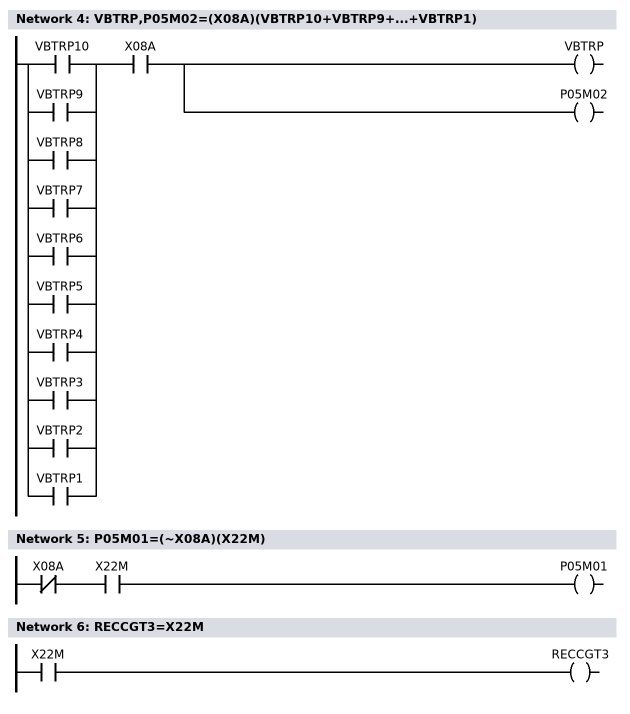
NETWORK
TITLE = VBTRP,P05M02=(X08A)(VBTRP10+VBTRP9+...+VBTRP1)
      A(;
      O     "VBTRP10";
      O     "VBTRP9";
      O     "VBTRP8";
      O     "VBTRP7";
      O     "VBTRP6";
      O     "VBTRP5";
      O     "VBTRP4";
      O     "VBTRP3";
      O     "VBTRP2";
      O     "VBTRP1";
      );
      A     "X08A";
      =     "VBTRP";
      =     "P05M02";
NETWORK
TITLE = P05M01=(~X08A)(X22M)
      AN    "X08A";
      A     "X22M";
      =     "P05M01";
NETWORK
TITLE = RECCGT3=X22M
      A     "X22M";
      =     "RECCGT3";
END_FUNCTION

FUNCTION "Sheet 22 (ATC)" : VOID	// FC 101
TITLE = Sheet 22 (ATC)
//LADDERS 32, 33, 41. VIBRATION RUNUP / RUNDOWN LOGIC (Digital)
AUTHOR : RJ
FAMILY : ATC
VERSION : 0.1
BEGIN
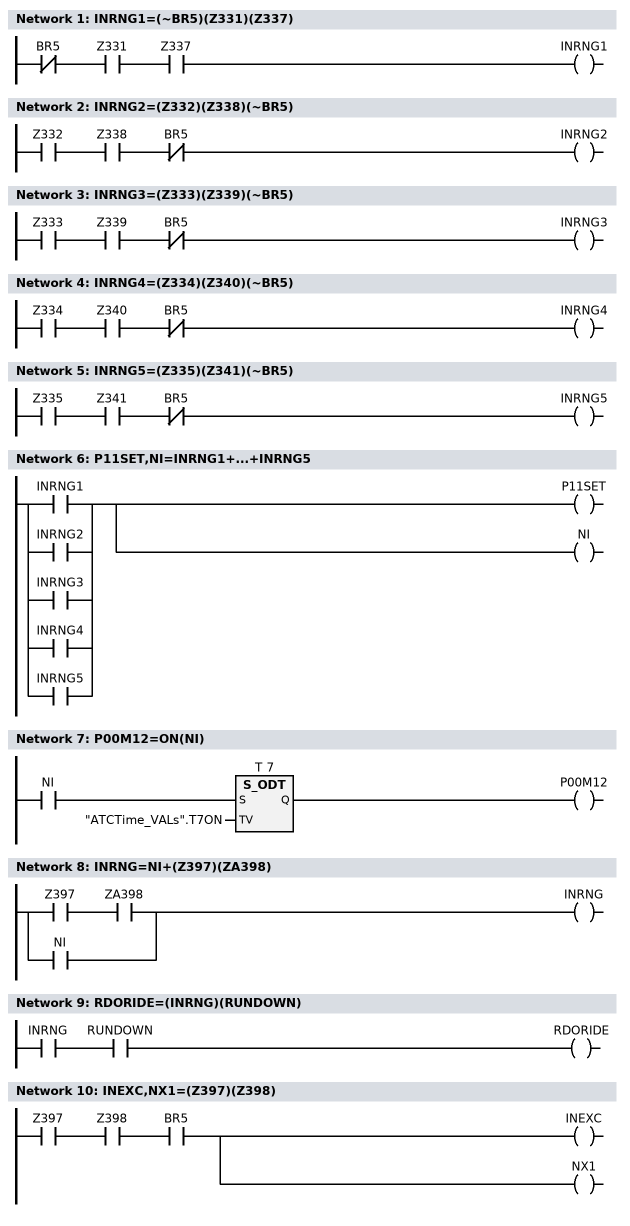
NETWORK
TITLE = INRNG1=(~BR5)(Z331)(Z337)
      AN    "BR5";
      A     "Z331";
      A     "Z337";
      =     "INRNG1";
NETWORK
TITLE = INRNG2=(Z332)(Z338)(~BR5)
      A     "Z332";
      A     "Z338";
      AN    "BR5";
      =     "INRNG2";
NETWORK
TITLE = INRNG3=(Z333)(Z339)(~BR5)
      A     "Z333";
      A     "Z339";
      AN    "BR5";
      =     "INRNG3";
NETWORK
TITLE = INRNG4=(Z334)(Z340)(~BR5)
      A     "Z334";
      A     "Z340";
      AN    "BR5";
      =     "INRNG4";
NETWORK
TITLE = INRNG5=(Z335)(Z341)(~BR5)
      A     "Z335";
      A     "Z341";
      AN    "BR5";
      =     "INRNG5";
NETWORK
TITLE = P11SET,NI=INRNG1+...+INRNG5
      O     "INRNG1";
      O     "INRNG2";
      O     "INRNG3";
      O     "INRNG4";
      O     "INRNG5";
      =     "P11SET";
      =     "NI";
NETWORK
TITLE = P00M12=ON(NI)
      A     "NI";
      L     "ATCTime_VALs".T7ON;
      SD    T 7;
      NOP   0;
      NOP   0;
      NOP   0;
      A     T 7;
      =     "P00M12";
NETWORK
TITLE = INRNG=NI+(Z397)(ZA398)
      A     "Z397";
      A     "ZA398";
      O     "NI";
      =     "INRNG";
NETWORK
TITLE = RDORIDE=(INRNG)(RUNDOWN)
      A     "INRNG";
      A     "RUNDOWN";
      =     "RDORIDE";
NETWORK
TITLE = INEXC,NX1=(Z397)(Z398)
      A     "Z397";
      A     "Z398";
      A     "BR5";
      =     "INEXC";
      =     "NX1";
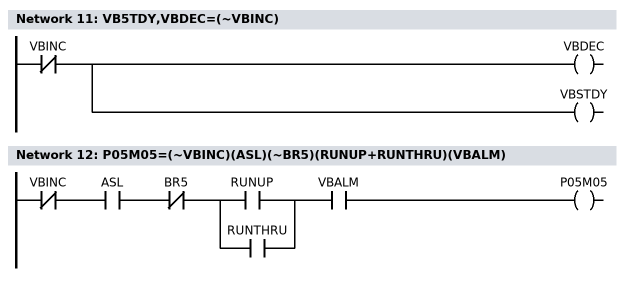
NETWORK
TITLE = VB5TDY,VBDEC=(~VBINC)
      AN    "VBINC";
      =     "VBDEC";
      =     "VBSTDY";
NETWORK
TITLE = P05M05=(~VBINC)(ASL)(~BR5)(RUNUP+RUNTHRU)(VBALM)
      AN    "VBINC";
      A     "ASL";
      AN    "BR5";
      A(;
      O     "RUNUP";
      O     "RUNTHRU";
      );
      A     "VBALM";
      =     "P05M05";
NETWORK
TITLE = HOLDSPD, HSOTIME
//HOLDSPD=FF[{(HSOTIME)(~INRNG)},{(~VBALM)+RUNUP+RUNTHRU+RUNDOWN+RUNBACK+VRSCNP}
//HSOTIME=FF{HOLSPD,(~VBALM)}
      A(;
      A     "HOLDSPD";
      S     "HSOTIME";
      AN    "VBALM";
      R     "HSOTIME";
      A     "HSOTIME";
      );
      AN    "INRNG";
      S     "HOLDSPD";
      A(;
      ON    "VBALM";
      O     "RUNUP";
      O     "RUNTHRU";
      O     "RUNDOWN";
      O     "RUNBACK";
      O     "VRSCNP";
      );
      R     "HOLDSPD";
      A     "HOLDSPD";
      =     "HOLDSPD";
END_FUNCTION

FUNCTION "Sheet 23 (ATC)" : VOID	// FC 102
TITLE = Sheet 23 (ATC)
//LADDER 39. VIBRATION RUNDOWN / RUNBACK LOGIC (Digital)
AUTHOR : RJ
FAMILY : ATC
VERSION : 0.1
BEGIN
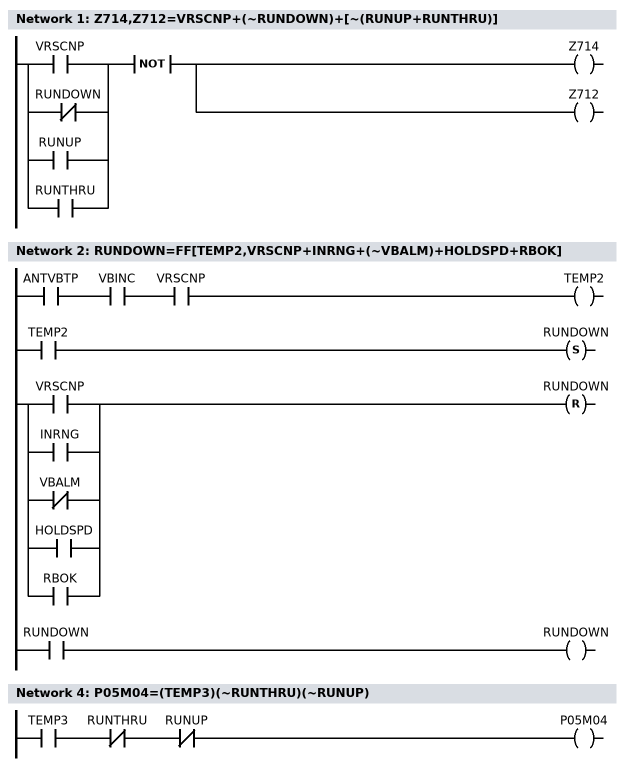
NETWORK
TITLE = Z714,Z712=VRSCNP+(~RUNDOWN)+[~(RUNUP+RUNTHRU)]
      O     "VRSCNP";
      ON    "RUNDOWN";
      O;
      A(;
      O     "RUNUP";
      O     "RUNTHRU";
      );
      NOT;
      =     "Z714";
      =     "Z712";
NETWORK
TITLE = RUNDOWN=FF[TEMP2,VRSCNP+INRNG+(~VBALM)+HOLDSPD+RBOK]
//TEMP2=(ANTVBTP)(VBINC)(VRSCNP)
      A     "ANTVBTP";
      A     "VBINC";
      A     "VRSCNP";
      =     "TEMP2";
      A     "TEMP2";
      S     "RUNDOWN";
      A(;
      O     "VRSCNP";
      O     "INRNG";
      ON    "VBALM";
      O     "HOLDSPD";
      O     "RBOK";
      );
      R     "RUNDOWN";
      A     "RUNDOWN";
      =     "RUNDOWN";
NETWORK
TITLE = RUNBACK, TEMP3
//RUNBACK=[(TEMP2)(~HOLDSPD)(RBOK)(~INRNG)(VBALM)]+FF[TEMP3,VRSCNP+RUNDOWN
//+RUNTHRU+RUNUP+(~RDEQASR)]
//TEMP3=RDORIDE+(HLDWS+VBALM+REQTRIP)(INEXC+INRNG)
      A     "TEMP2";
      AN    "HOLDSPD";
      A     "RBOK";
      AN    "INRNG";
      A     "VBALM";
      O(;
      A(;
      O     "RDORIDE";
      O;
      A(;
      O     "HLDWS";
      O     "VBALM";
      O     "REQTRIP";
      );
      A(;
      O     "INEXC";
      O     "INRNG";
      );
      );
      =     "TEMP3";
      A     "TEMP3";
      S     "TEMP4";
      A(;
      O     "VRSCNP";
      O     "RUNDOWN";
      O     "RUNTHRU";
      O     "RUNUP";
      ON    "RDEQASR";
      );
      R     "TEMP4";
      A     "TEMP4";
      );
      =     "RUNBACK";
NETWORK
TITLE = P05M04=(TEMP3)(~RUNTHRU)(~RUNUP)
      A     "TEMP3";
      AN    "RUNTHRU";
      AN    "RUNUP";
      =     "P05M04";
END_FUNCTION

FUNCTION "3xHISIGMTV, 1xLOSIGMTV" : VOID	// FC 103
TITLE = 3xHISIGMTV, 1xLOSIGMTV
AUTHOR : RJ
VERSION : 0.1
VAR_INPUT
  IN_HI1 : REAL ;
  IN_HI2 : REAL ;
  IN_HI3 : REAL ;
  IN_LO : REAL ;
  STPT : REAL ;
  Param_HI1 : UDT 8;
  Param_HI2 : UDT 8;
  Param_HI3 : UDT 8;
  Param_LO : UDT 9;
END_VAR
VAR_OUTPUT
  OUT_HI1 : BOOL ;
  OUT_HI2 : BOOL ;
  OUT_HI3 : BOOL ;
  OUT_LO : BOOL ;
END_VAR
VAR_TEMP
  TEMP_HI1 : UDT 8;
  TEMP_HI2 : UDT 8;
  TEMP_HI3 : UDT 8;
  TEMP_LO : UDT 9;
END_VAR
BEGIN
NETWORK
TITLE =
      BLD   5;
      T     LD 18;
      TAK;
      T     LD 22;
      L     P##Param_HI1;
      LAR1;
      L     W [AR1,P#0.0];
      T     LW 16;
      OPN   DB [LW 16];
      L     D [AR1,P#2.0];
      LAR1;
      L     LD 22;
      L     LD 18;
      L     D [AR1,P#0.0];
      T     #TEMP_HI1;
      NOP   0;
NETWORK
TITLE =
      BLD   5;
      T     LD 18;
      TAK;
      T     LD 22;
      L     P##Param_HI2;
      LAR1;
      L     W [AR1,P#0.0];
      T     LW 16;
      OPN   DB [LW 16];
      L     D [AR1,P#2.0];
      LAR1;
      L     LD 22;
      L     LD 18;
      L     D [AR1,P#0.0];
      T     #TEMP_HI2;
      NOP   0;
NETWORK
TITLE =
      BLD   5;
      T     LD 18;
      TAK;
      T     LD 22;
      L     P##Param_HI3;
      LAR1;
      L     W [AR1,P#0.0];
      T     LW 16;
      OPN   DB [LW 16];
      L     D [AR1,P#2.0];
      LAR1;
      L     LD 22;
      L     LD 18;
      L     D [AR1,P#0.0];
      T     #TEMP_HI3;
      NOP   0;
NETWORK
TITLE =
      BLD   5;
      T     LD 18;
      TAK;
      T     LD 22;
      L     P##Param_LO;
      LAR1;
      L     W [AR1,P#0.0];
      T     LW 16;
      OPN   DB [LW 16];
      L     D [AR1,P#2.0];
      LAR1;
      L     LD 22;
      L     LD 18;
      L     D [AR1,P#0.0];
      T     #TEMP_LO;
      NOP   0;
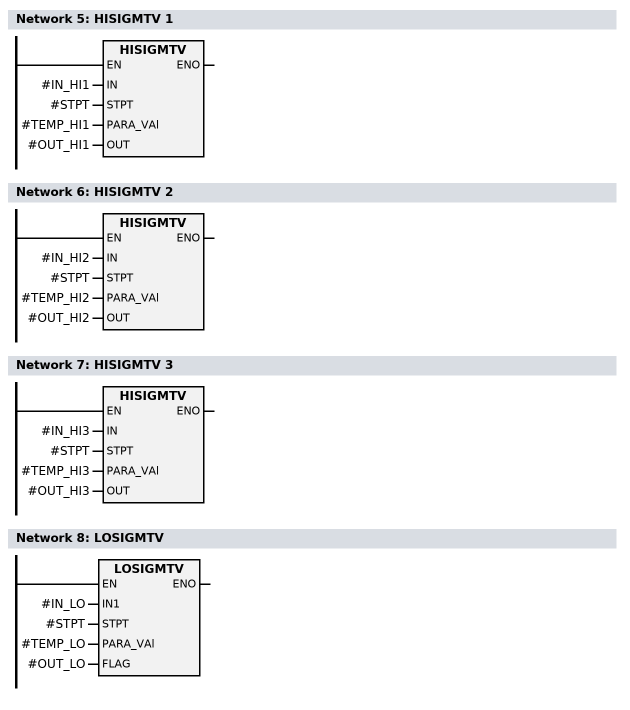
NETWORK
TITLE = HISIGMTV 1
      CALL  "HISIGMTV" (
           IN                       := #IN_HI1,
           STPT                     := #STPT,
           PARA_VAl                 := #TEMP_HI1,
           OUT                      := #OUT_HI1);
      NOP   0;
NETWORK
TITLE = HISIGMTV 2
      CALL  "HISIGMTV" (
           IN                       := #IN_HI2,
           STPT                     := #STPT,
           PARA_VAl                 := #TEMP_HI2,
           OUT                      := #OUT_HI2);
      NOP   0;
NETWORK
TITLE = HISIGMTV 3
      CALL  "HISIGMTV" (
           IN                       := #IN_HI3,
           STPT                     := #STPT,
           PARA_VAl                 := #TEMP_HI3,
           OUT                      := #OUT_HI3);
      NOP   0;
NETWORK
TITLE = LOSIGMTV
      CALL  "LOSIGMTV" (
           IN1                      := #IN_LO,
           STPT                     := #STPT,
           PARA_VAl                 := #TEMP_LO,
           FLAG                     := #OUT_LO);
      NOP   0;
END_FUNCTION

FUNCTION "3xLOSIGMTV, 1xHISIGMTV" : VOID	// FC 104
TITLE = 3xLOSIGMTV, 1xHISIGMTV
AUTHOR : RJ
VERSION : 0.1
VAR_INPUT
  IN_LO1 : REAL ;
  IN_LO2 : REAL ;
  IN_LO3 : REAL ;
  IN_HI : REAL ;
  STPT : REAL ;
  Param_LO1 : UDT 9;
  Param_LO2 : UDT 9;
  Param_LO3 : UDT 9;
  Param_HI : UDT 8;
END_VAR
VAR_OUTPUT
  OUT_LO1 : BOOL ;
  OUT_LO2 : BOOL ;
  OUT_LO3 : BOOL ;
  OUT_HI : BOOL ;
END_VAR
VAR_TEMP
  TEMP_LO1 : UDT 9;
  TEMP_LO2 : UDT 9;
  TEMP_LO3 : UDT 9;
  TEMP_HI : UDT 8;
END_VAR
BEGIN
NETWORK
TITLE =
      BLD   5;
      T     LD 18;
      TAK;
      T     LD 22;
      L     P##Param_LO1;
      LAR1;
      L     W [AR1,P#0.0];
      T     LW 16;
      OPN   DB [LW 16];
      L     D [AR1,P#2.0];
      LAR1;
      L     LD 22;
      L     LD 18;
      L     D [AR1,P#0.0];
      T     #TEMP_LO1;
      NOP   0;
NETWORK
TITLE =
      BLD   5;
      T     LD 18;
      TAK;
      T     LD 22;
      L     P##Param_LO2;
      LAR1;
      L     W [AR1,P#0.0];
      T     LW 16;
      OPN   DB [LW 16];
      L     D [AR1,P#2.0];
      LAR1;
      L     LD 22;
      L     LD 18;
      L     D [AR1,P#0.0];
      T     #TEMP_LO2;
      NOP   0;
NETWORK
TITLE =
      BLD   5;
      T     LD 18;
      TAK;
      T     LD 22;
      L     P##Param_LO3;
      LAR1;
      L     W [AR1,P#0.0];
      T     LW 16;
      OPN   DB [LW 16];
      L     D [AR1,P#2.0];
      LAR1;
      L     LD 22;
      L     LD 18;
      L     D [AR1,P#0.0];
      T     #TEMP_LO3;
      NOP   0;
NETWORK
TITLE =
      BLD   5;
      T     LD 18;
      TAK;
      T     LD 22;
      L     P##Param_HI;
      LAR1;
      L     W [AR1,P#0.0];
      T     LW 16;
      OPN   DB [LW 16];
      L     D [AR1,P#2.0];
      LAR1;
      L     LD 22;
      L     LD 18;
      L     D [AR1,P#0.0];
      T     #TEMP_HI;
      NOP   0;
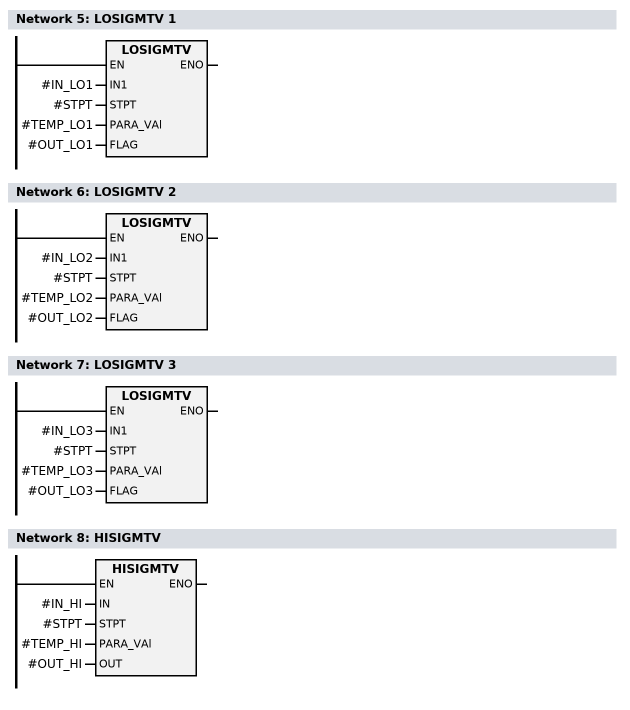
NETWORK
TITLE = LOSIGMTV 1
      CALL  "LOSIGMTV" (
           IN1                      := #IN_LO1,
           STPT                     := #STPT,
           PARA_VAl                 := #TEMP_LO1,
           FLAG                     := #OUT_LO1);
      NOP   0;
NETWORK
TITLE = LOSIGMTV 2
      CALL  "LOSIGMTV" (
           IN1                      := #IN_LO2,
           STPT                     := #STPT,
           PARA_VAl                 := #TEMP_LO2,
           FLAG                     := #OUT_LO2);
      NOP   0;
NETWORK
TITLE = LOSIGMTV 3
      CALL  "LOSIGMTV" (
           IN1                      := #IN_LO3,
           STPT                     := #STPT,
           PARA_VAl                 := #TEMP_LO3,
           FLAG                     := #OUT_LO3);
      NOP   0;
NETWORK
TITLE = HISIGMTV
      CALL  "HISIGMTV" (
           IN                       := #IN_HI,
           STPT                     := #STPT,
           PARA_VAl                 := #TEMP_HI,
           OUT                      := #OUT_HI);
      NOP   0;
END_FUNCTION

// FC 105: know-how protected block, not included

FUNCTION "Sheet 25 (ATC)" : VOID	// FC 106
TITLE = Sheet 25 (ATC)
//SPEED RESONANT RANGE MONITOR (Analog)
AUTHOR : RJ
FAMILY : ATC
VERSION : 0.1
BEGIN
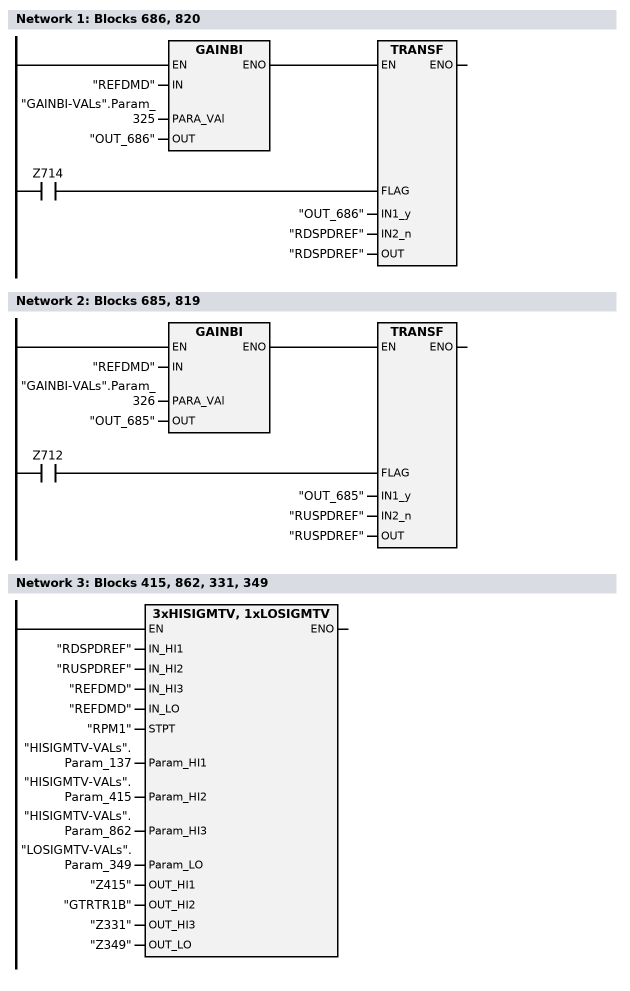
NETWORK
TITLE = Blocks 686, 820
      A     "Z714";
      =     L 0.0;
      BLD   103;
      A(;
      CALL  "GAINBI" (
           IN                       := "REFDMD",
           PARA_VAl                 := "GAINBI-VALs".Param_325,
           OUT                      := "OUT_686");
      A     BR;
      );
      JNB   _001;
      CALL  "TRANSF" (
           FLAG                     := L 0.0,
           IN1_y                    := "OUT_686",
           IN2_n                    := "RDSPDREF",
           OUT                      := "RDSPDREF");
_001: NOP   0;
NETWORK
TITLE = Blocks 685, 819
      A     "Z712";
      =     L 0.0;
      BLD   103;
      A(;
      CALL  "GAINBI" (
           IN                       := "REFDMD",
           PARA_VAl                 := "GAINBI-VALs".Param_326,
           OUT                      := "OUT_685");
      A     BR;
      );
      JNB   _002;
      CALL  "TRANSF" (
           FLAG                     := L 0.0,
           IN1_y                    := "OUT_685",
           IN2_n                    := "RUSPDREF",
           OUT                      := "RUSPDREF");
_002: NOP   0;
NETWORK
TITLE = Blocks 415, 862, 331, 349
      CALL  "3xHISIGMTV, 1xLOSIGMTV" (
           IN_HI1                   := "RDSPDREF",
           IN_HI2                   := "RUSPDREF",
           IN_HI3                   := "REFDMD",
           IN_LO                    := "REFDMD",
           STPT                     := "RPM1",
           Param_HI1                := "HISIGMTV-VALs".Param_137,
           Param_HI2                := "HISIGMTV-VALs".Param_415,
           Param_HI3                := "HISIGMTV-VALs".Param_862,
           Param_LO                 := "LOSIGMTV-VALs".Param_349,
           OUT_HI1                  := "Z415",
           OUT_HI2                  := "GTRTR1B",
           OUT_HI3                  := "Z331",
           OUT_LO                   := "Z349");
      NOP   0;
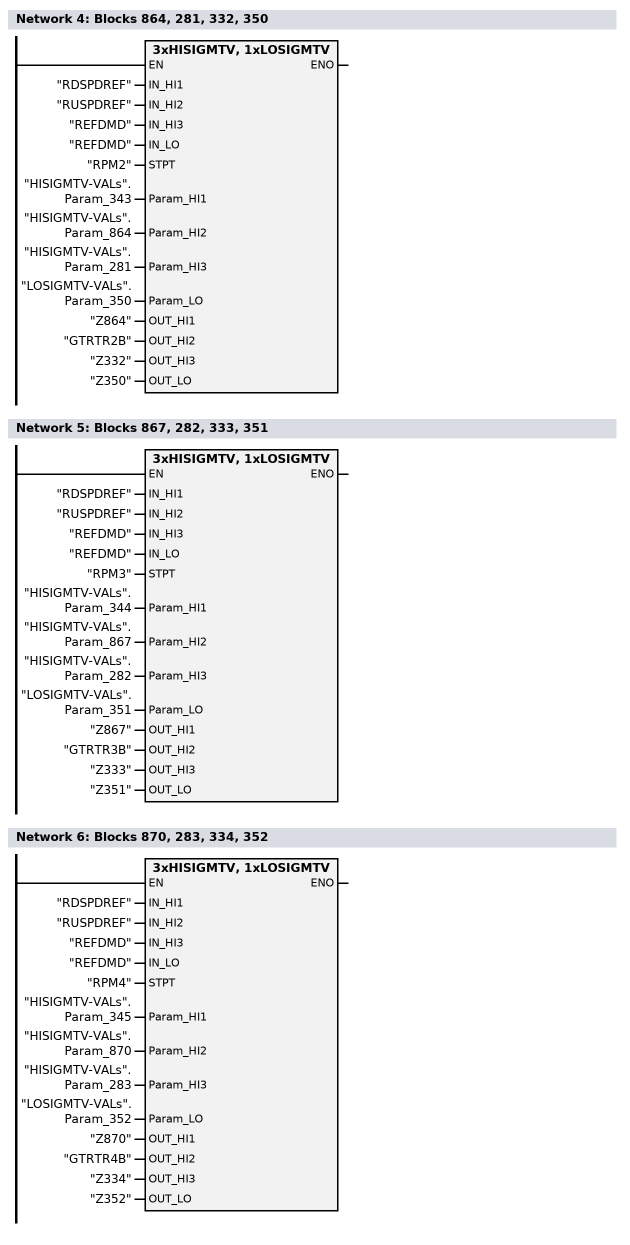
NETWORK
TITLE = Blocks 864, 281, 332, 350
      CALL  "3xHISIGMTV, 1xLOSIGMTV" (
           IN_HI1                   := "RDSPDREF",
           IN_HI2                   := "RUSPDREF",
           IN_HI3                   := "REFDMD",
           IN_LO                    := "REFDMD",
           STPT                     := "RPM2",
           Param_HI1                := "HISIGMTV-VALs".Param_343,
           Param_HI2                := "HISIGMTV-VALs".Param_864,
           Param_HI3                := "HISIGMTV-VALs".Param_281,
           Param_LO                 := "LOSIGMTV-VALs".Param_350,
           OUT_HI1                  := "Z864",
           OUT_HI2                  := "GTRTR2B",
           OUT_HI3                  := "Z332",
           OUT_LO                   := "Z350");
      NOP   0;
NETWORK
TITLE = Blocks 867, 282, 333, 351
      CALL  "3xHISIGMTV, 1xLOSIGMTV" (
           IN_HI1                   := "RDSPDREF",
           IN_HI2                   := "RUSPDREF",
           IN_HI3                   := "REFDMD",
           IN_LO                    := "REFDMD",
           STPT                     := "RPM3",
           Param_HI1                := "HISIGMTV-VALs".Param_344,
           Param_HI2                := "HISIGMTV-VALs".Param_867,
           Param_HI3                := "HISIGMTV-VALs".Param_282,
           Param_LO                 := "LOSIGMTV-VALs".Param_351,
           OUT_HI1                  := "Z867",
           OUT_HI2                  := "GTRTR3B",
           OUT_HI3                  := "Z333",
           OUT_LO                   := "Z351");
      NOP   0;
NETWORK
TITLE = Blocks 870, 283, 334, 352
      CALL  "3xHISIGMTV, 1xLOSIGMTV" (
           IN_HI1                   := "RDSPDREF",
           IN_HI2                   := "RUSPDREF",
           IN_HI3                   := "REFDMD",
           IN_LO                    := "REFDMD",
           STPT                     := "RPM4",
           Param_HI1                := "HISIGMTV-VALs".Param_345,
           Param_HI2                := "HISIGMTV-VALs".Param_870,
           Param_HI3                := "HISIGMTV-VALs".Param_283,
           Param_LO                 := "LOSIGMTV-VALs".Param_352,
           OUT_HI1                  := "Z870",
           OUT_HI2                  := "GTRTR4B",
           OUT_HI3                  := "Z334",
           OUT_LO                   := "Z352");
      NOP   0;
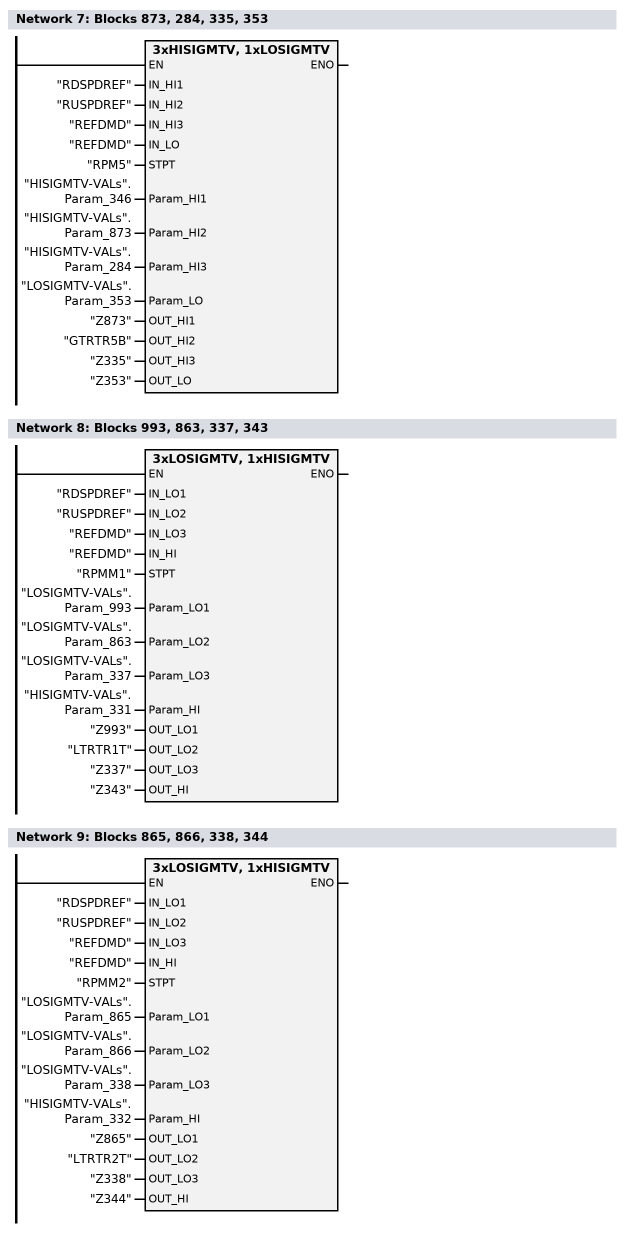
NETWORK
TITLE = Blocks 873, 284, 335, 353
      CALL  "3xHISIGMTV, 1xLOSIGMTV" (
           IN_HI1                   := "RDSPDREF",
           IN_HI2                   := "RUSPDREF",
           IN_HI3                   := "REFDMD",
           IN_LO                    := "REFDMD",
           STPT                     := "RPM5",
           Param_HI1                := "HISIGMTV-VALs".Param_346,
           Param_HI2                := "HISIGMTV-VALs".Param_873,
           Param_HI3                := "HISIGMTV-VALs".Param_284,
           Param_LO                 := "LOSIGMTV-VALs".Param_353,
           OUT_HI1                  := "Z873",
           OUT_HI2                  := "GTRTR5B",
           OUT_HI3                  := "Z335",
           OUT_LO                   := "Z353");
      NOP   0;
NETWORK
TITLE = Blocks 993, 863, 337, 343
      CALL  "3xLOSIGMTV, 1xHISIGMTV" (
           IN_LO1                   := "RDSPDREF",
           IN_LO2                   := "RUSPDREF",
           IN_LO3                   := "REFDMD",
           IN_HI                    := "REFDMD",
           STPT                     := "RPMM1",
           Param_LO1                := "LOSIGMTV-VALs".Param_993,
           Param_LO2                := "LOSIGMTV-VALs".Param_863,
           Param_LO3                := "LOSIGMTV-VALs".Param_337,
           Param_HI                 := "HISIGMTV-VALs".Param_331,
           OUT_LO1                  := "Z993",
           OUT_LO2                  := "LTRTR1T",
           OUT_LO3                  := "Z337",
           OUT_HI                   := "Z343");
      NOP   0;
NETWORK
TITLE = Blocks 865, 866, 338, 344
      CALL  "3xLOSIGMTV, 1xHISIGMTV" (
           IN_LO1                   := "RDSPDREF",
           IN_LO2                   := "RUSPDREF",
           IN_LO3                   := "REFDMD",
           IN_HI                    := "REFDMD",
           STPT                     := "RPMM2",
           Param_LO1                := "LOSIGMTV-VALs".Param_865,
           Param_LO2                := "LOSIGMTV-VALs".Param_866,
           Param_LO3                := "LOSIGMTV-VALs".Param_338,
           Param_HI                 := "HISIGMTV-VALs".Param_332,
           OUT_LO1                  := "Z865",
           OUT_LO2                  := "LTRTR2T",
           OUT_LO3                  := "Z338",
           OUT_HI                   := "Z344");
      NOP   0;
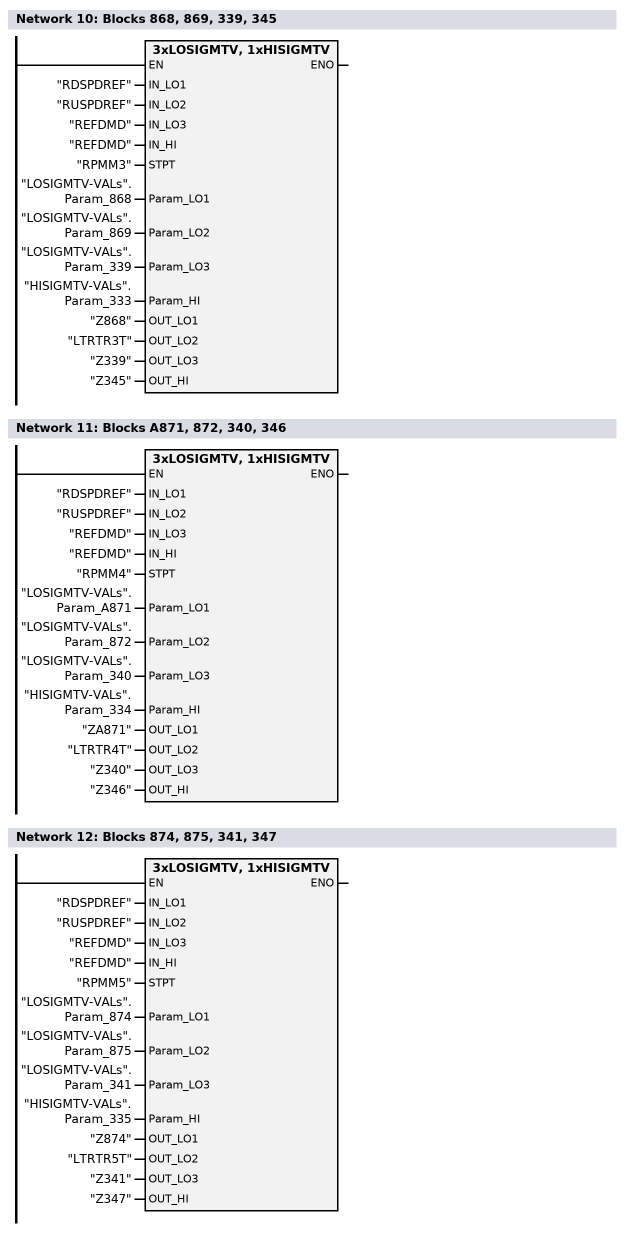
NETWORK
TITLE = Blocks 868, 869, 339, 345
      CALL  "3xLOSIGMTV, 1xHISIGMTV" (
           IN_LO1                   := "RDSPDREF",
           IN_LO2                   := "RUSPDREF",
           IN_LO3                   := "REFDMD",
           IN_HI                    := "REFDMD",
           STPT                     := "RPMM3",
           Param_LO1                := "LOSIGMTV-VALs".Param_868,
           Param_LO2                := "LOSIGMTV-VALs".Param_869,
           Param_LO3                := "LOSIGMTV-VALs".Param_339,
           Param_HI                 := "HISIGMTV-VALs".Param_333,
           OUT_LO1                  := "Z868",
           OUT_LO2                  := "LTRTR3T",
           OUT_LO3                  := "Z339",
           OUT_HI                   := "Z345");
      NOP   0;
NETWORK
TITLE = Blocks A871, 872, 340, 346
      CALL  "3xLOSIGMTV, 1xHISIGMTV" (
           IN_LO1                   := "RDSPDREF",
           IN_LO2                   := "RUSPDREF",
           IN_LO3                   := "REFDMD",
           IN_HI                    := "REFDMD",
           STPT                     := "RPMM4",
           Param_LO1                := "LOSIGMTV-VALs".Param_A871,
           Param_LO2                := "LOSIGMTV-VALs".Param_872,
           Param_LO3                := "LOSIGMTV-VALs".Param_340,
           Param_HI                 := "HISIGMTV-VALs".Param_334,
           OUT_LO1                  := "ZA871",
           OUT_LO2                  := "LTRTR4T",
           OUT_LO3                  := "Z340",
           OUT_HI                   := "Z346");
      NOP   0;
NETWORK
TITLE = Blocks 874, 875, 341, 347
      CALL  "3xLOSIGMTV, 1xHISIGMTV" (
           IN_LO1                   := "RDSPDREF",
           IN_LO2                   := "RUSPDREF",
           IN_LO3                   := "REFDMD",
           IN_HI                    := "REFDMD",
           STPT                     := "RPMM5",
           Param_LO1                := "LOSIGMTV-VALs".Param_874,
           Param_LO2                := "LOSIGMTV-VALs".Param_875,
           Param_LO3                := "LOSIGMTV-VALs".Param_341,
           Param_HI                 := "HISIGMTV-VALs".Param_335,
           OUT_LO1                  := "Z874",
           OUT_LO2                  := "LTRTR5T",
           OUT_LO3                  := "Z341",
           OUT_HI                   := "Z347");
      NOP   0;
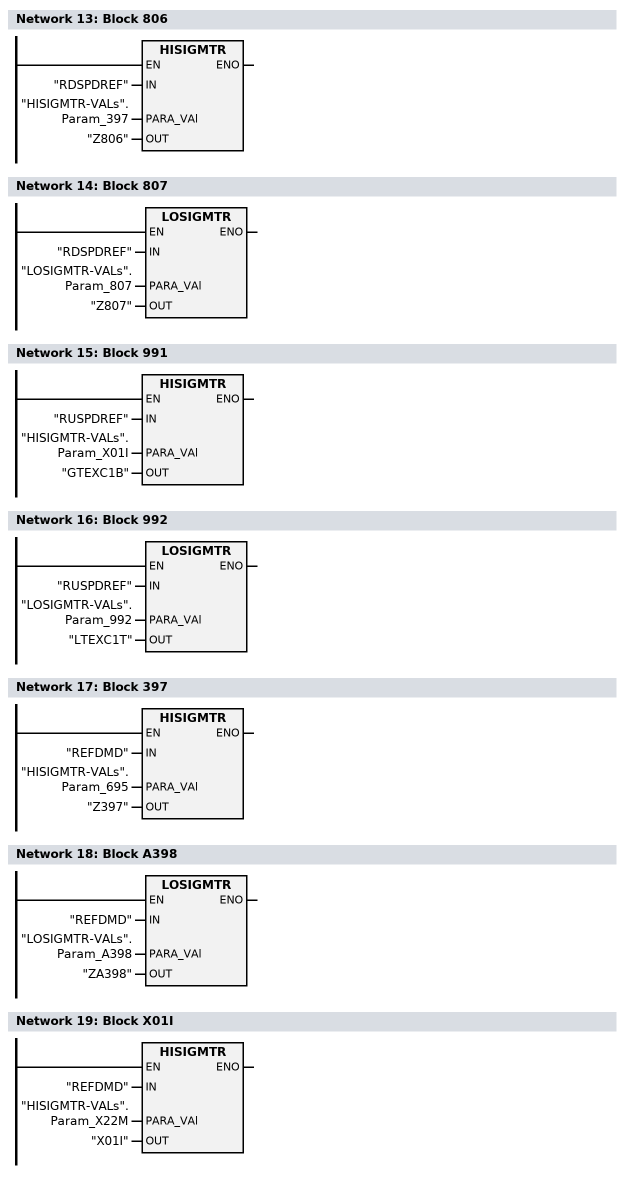
NETWORK
TITLE = Block 806
      CALL  "HISIGMTR" (
           IN                       := "RDSPDREF",
           PARA_VAl                 := "HISIGMTR-VALs".Param_397,
           OUT                      := "Z806");
      NOP   0;
NETWORK
TITLE = Block 807
      CALL  "LOSIGMTR" (
           IN                       := "RDSPDREF",
           PARA_VAl                 := "LOSIGMTR-VALs".Param_807,
           OUT                      := "Z807");
      NOP   0;
NETWORK
TITLE = Block 991
      CALL  "HISIGMTR" (
           IN                       := "RUSPDREF",
           PARA_VAl                 := "HISIGMTR-VALs".Param_X01I,
           OUT                      := "GTEXC1B");
      NOP   0;
NETWORK
TITLE = Block 992
      CALL  "LOSIGMTR" (
           IN                       := "RUSPDREF",
           PARA_VAl                 := "LOSIGMTR-VALs".Param_992,
           OUT                      := "LTEXC1T");
      NOP   0;
NETWORK
TITLE = Block 397
      CALL  "HISIGMTR" (
           IN                       := "REFDMD",
           PARA_VAl                 := "HISIGMTR-VALs".Param_695,
           OUT                      := "Z397");
      NOP   0;
NETWORK
TITLE = Block A398
      CALL  "LOSIGMTR" (
           IN                       := "REFDMD",
           PARA_VAl                 := "LOSIGMTR-VALs".Param_A398,
           OUT                      := "ZA398");
      NOP   0;
NETWORK
TITLE = Block X01I
      CALL  "HISIGMTR" (
           IN                       := "REFDMD",
           PARA_VAl                 := "HISIGMTR-VALs".Param_X22M,
           OUT                      := "X01I");
      NOP   0;
END_FUNCTION

FUNCTION "Sheet 26 (ATC)" : VOID	// FC 107
TITLE = Sheet 26 (ATC)
//LADDERS 150, 420. VIBRATION SPEED REF LOGIC (Digital)
AUTHOR : RJ
FAMILY : ATC
VERSION : 0.1
BEGIN
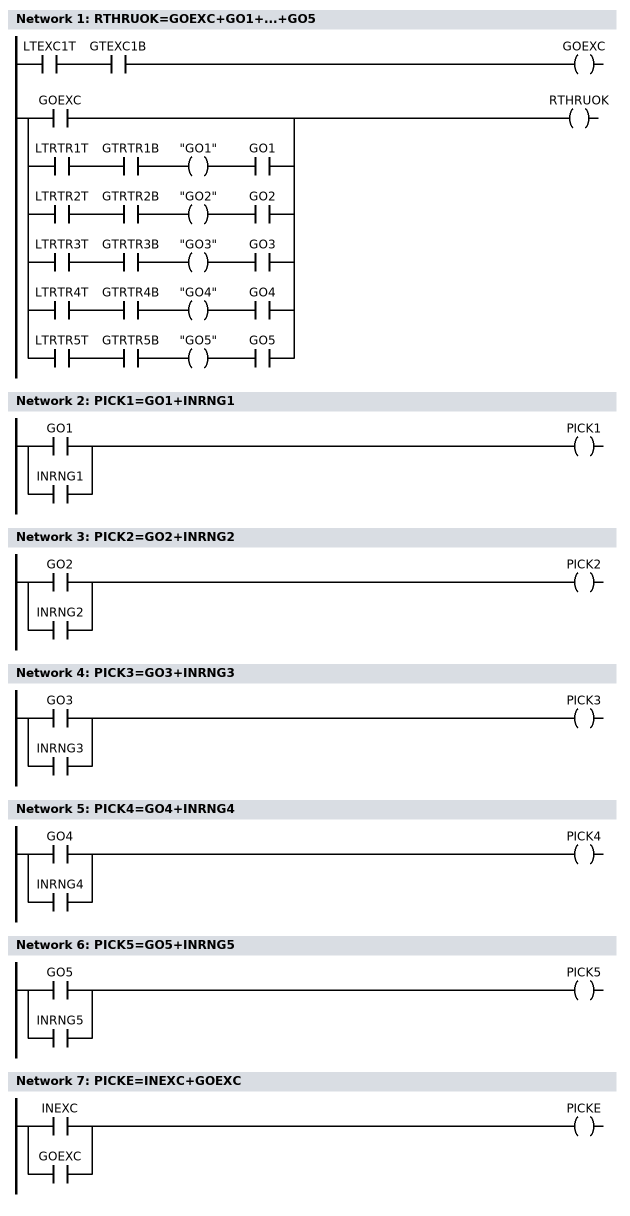
NETWORK
TITLE = RTHRUOK=GOEXC+GO1+...+GO5
//GOEXC=(LTEXC1T)(GTEXC1B)
//GO1=(LTRTR1T)(GTRTR1B)
//...
//GO5=(LTRTR5T)(GTRTR5B)
      A     "LTEXC1T";
      A     "GTEXC1B";
      =     "GOEXC";
      A     "GOEXC";
      O(;
      A     "LTRTR1T";
      A     "GTRTR1B";
      =     "GO1";
      A     "GO1";
      );
      O(;
      A     "LTRTR2T";
      A     "GTRTR2B";
      =     "GO2";
      A     "GO2";
      );
      O(;
      A     "LTRTR3T";
      A     "GTRTR3B";
      =     "GO3";
      A     "GO3";
      );
      O(;
      A     "LTRTR4T";
      A     "GTRTR4B";
      =     "GO4";
      A     "GO4";
      );
      O(;
      A     "LTRTR5T";
      A     "GTRTR5B";
      =     "GO5";
      A     "GO5";
      );
      =     "RTHRUOK";
NETWORK
TITLE = PICK1=GO1+INRNG1
      O     "GO1";
      O     "INRNG1";
      =     "PICK1";
NETWORK
TITLE = PICK2=GO2+INRNG2
      O     "GO2";
      O     "INRNG2";
      =     "PICK2";
NETWORK
TITLE = PICK3=GO3+INRNG3
      O     "GO3";
      O     "INRNG3";
      =     "PICK3";
NETWORK
TITLE = PICK4=GO4+INRNG4
      O     "GO4";
      O     "INRNG4";
      =     "PICK4";
NETWORK
TITLE = PICK5=GO5+INRNG5
      O     "GO5";
      O     "INRNG5";
      =     "PICK5";
NETWORK
TITLE = PICKE=INEXC+GOEXC
      O     "INEXC";
      O     "GOEXC";
      =     "PICKE";
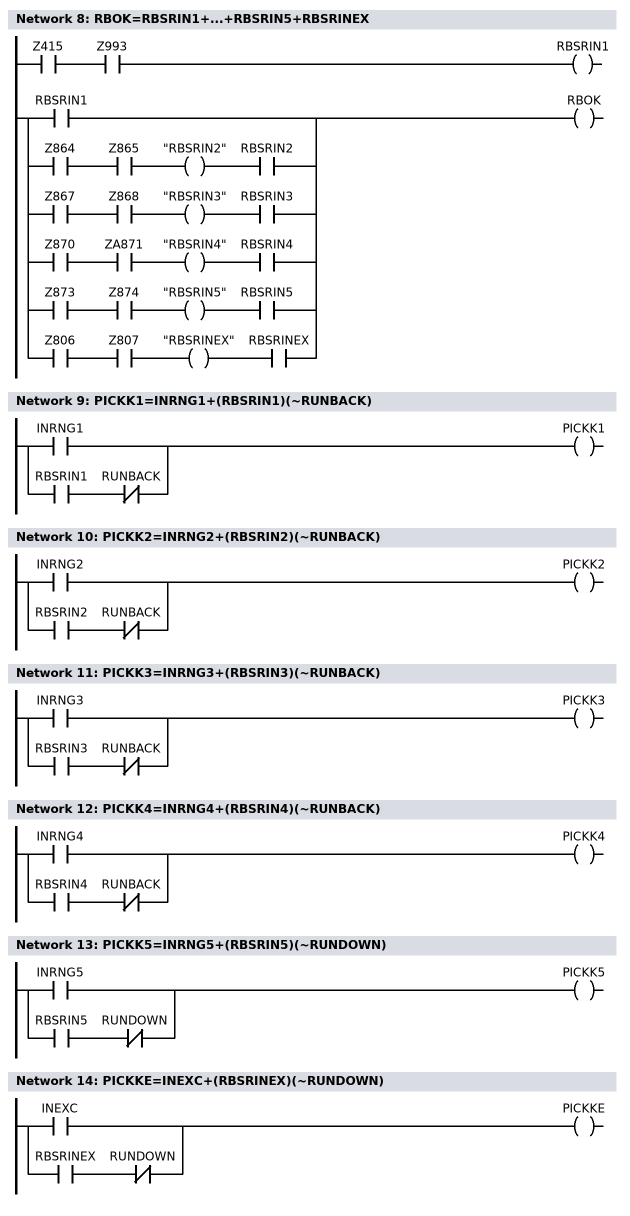
NETWORK
TITLE = RBOK=RBSRIN1+...+RBSRIN5+RBSRINEX
//RBSRIN1=(Z415)(Z993)
//RBSRIN2=(Z864)(Z865)
//RBSRIN3=(Z867)(Z868)
//RBSRIN4=(Z870)(ZA871)
//RBSRIN5=(Z873)(Z874)
//RBSRINEX=(Z806)(Z807)
      A     "Z415";
      A     "Z993";
      =     "RBSRIN1";
      A     "RBSRIN1";
      O(;
      A     "Z864";
      A     "Z865";
      =     "RBSRIN2";
      A     "RBSRIN2";
      );
      O(;
      A     "Z867";
      A     "Z868";
      =     "RBSRIN3";
      A     "RBSRIN3";
      );
      O(;
      A     "Z870";
      A     "ZA871";
      =     "RBSRIN4";
      A     "RBSRIN4";
      );
      O(;
      A     "Z873";
      A     "Z874";
      =     "RBSRIN5";
      A     "RBSRIN5";
      );
      O(;
      A     "Z806";
      A     "Z807";
      =     "RBSRINEX";
      A     "RBSRINEX";
      );
      =     "RBOK";
NETWORK
TITLE = PICKK1=INRNG1+(RBSRIN1)(~RUNBACK)
      O     "INRNG1";
      O;
      A     "RBSRIN1";
      AN    "RUNBACK";
      =     "PICKK1";
NETWORK
TITLE = PICKK2=INRNG2+(RBSRIN2)(~RUNBACK)
      O     "INRNG2";
      O;
      A     "RBSRIN2";
      AN    "RUNBACK";
      =     "PICKK2";
NETWORK
TITLE = PICKK3=INRNG3+(RBSRIN3)(~RUNBACK)
      O     "INRNG3";
      O;
      A     "RBSRIN3";
      AN    "RUNBACK";
      =     "PICKK3";
NETWORK
TITLE = PICKK4=INRNG4+(RBSRIN4)(~RUNBACK)
      O     "INRNG4";
      O;
      A     "RBSRIN4";
      AN    "RUNBACK";
      =     "PICKK4";
NETWORK
TITLE = PICKK5=INRNG5+(RBSRIN5)(~RUNDOWN)
      O     "INRNG5";
      O;
      A     "RBSRIN5";
      AN    "RUNDOWN";
      =     "PICKK5";
NETWORK
TITLE = PICKKE=INEXC+(RBSRINEX)(~RUNDOWN)
      O     "INEXC";
      O;
      A     "RBSRINEX";
      AN    "RUNDOWN";
      =     "PICKKE";
END_FUNCTION

FUNCTION "Sheet 27 (ATC)" : VOID	// FC 108
TITLE = Sheet 27 (ATC)
//VIBRATION RUNBACK SPEED REF (Analog)
AUTHOR : RJ
FAMILY : ATC
VERSION : 0.1
BEGIN
NETWORK
TITLE = Blocks 670, 671, 672
      A     "PICKK3";
      =     L 0.0;
      BLD   103;
      A(;
      A     "PICKK2";
      =     L 0.1;
      BLD   103;
      A(;
      A     "PICKK1";
      =     L 0.2;
      BLD   103;
      CALL  "TRANSF" (
           FLAG                     := L 0.2,
           IN1_y                    := "REFF1",
           IN2_n                    := "RBSPDREF",
           OUT                      := "OUT_670");
      A     BR;
      );
      JNB   _001;
      CALL  "TRANSF" (
           FLAG                     := L 0.1,
           IN1_y                    := "REFF2",
           IN2_n                    := "OUT_670",
           OUT                      := "OUT_671");
_001: A     BR;
      );
      JNB   _002;
      CALL  "TRANSF" (
           FLAG                     := L 0.0,
           IN1_y                    := "REFF3",
           IN2_n                    := "OUT_671",
           OUT                      := "OUT_672");
_002: NOP   0;
NETWORK
TITLE = Blocks 673, 674, 676
      A     "PICKKE";
      =     L 0.0;
      BLD   103;
      A(;
      A     "PICKK5";
      =     L 0.1;
      BLD   103;
      A(;
      A     "PICKK4";
      =     L 0.2;
      BLD   103;
      CALL  "TRANSF" (
           FLAG                     := L 0.2,
           IN1_y                    := "REFF4",
           IN2_n                    := "OUT_672",
           OUT                      := "OUT_673");
      A     BR;
      );
      JNB   _003;
      CALL  "TRANSF" (
           FLAG                     := L 0.1,
           IN1_y                    := "REFF5",
           IN2_n                    := "OUT_673",
           OUT                      := "OUT_674");
_003: A     BR;
      );
      JNB   _004;
      CALL  "TRANSF" (
           FLAG                     := L 0.0,
           IN1_y                    := "EXCREFF",
           IN2_n                    := "OUT_674",
           OUT                      := "RBSPDREF");
_004: NOP   0;
END_FUNCTION

FUNCTION "Sheet 28 (ATC)" : VOID	// FC 109
TITLE = Sheet 28 (ATC)
//LADDERS 30, 43, 307, 308, 309. VIBRATION RUNUP/RUNTHRU LOGIC (Digital)
AUTHOR : RJ
FAMILY : ATC
VERSION : 0.1
BEGIN
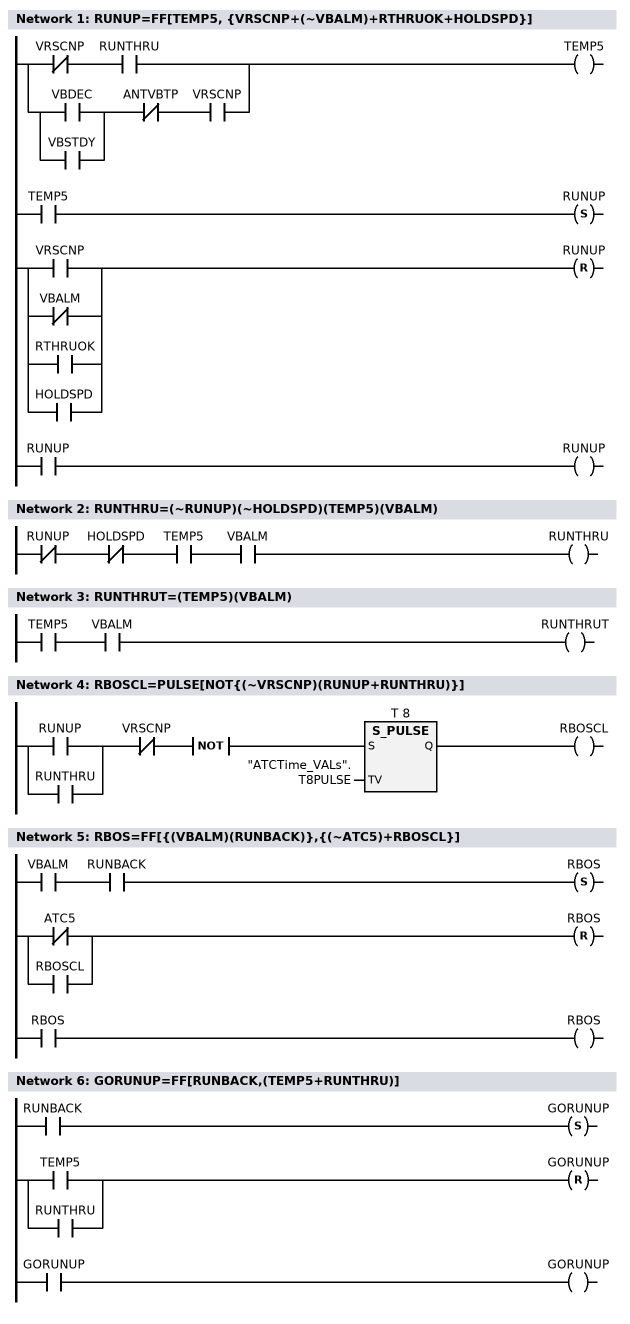
NETWORK
TITLE = RUNUP=FF[TEMP5, {VRSCNP+(~VBALM)+RTHRUOK+HOLDSPD}]
//TEMP5=[(~VRSCNP)(RUNTHRU)]+[(VBDEC+VBSTDY)(~ANTVBTP)(VRSCNP)]
      A(;
      AN    "VRSCNP";
      A     "RUNTHRU";
      O;
      A(;
      O     "VBDEC";
      O     "VBSTDY";
      );
      AN    "ANTVBTP";
      A     "VRSCNP";
      );
      =     "TEMP5";
      A     "TEMP5";
      S     "RUNUP";
      A(;
      O     "VRSCNP";
      ON    "VBALM";
      O     "RTHRUOK";
      O     "HOLDSPD";
      );
      R     "RUNUP";
      A     "RUNUP";
      =     "RUNUP";
NETWORK
TITLE = RUNTHRU=(~RUNUP)(~HOLDSPD)(TEMP5)(VBALM)
      AN    "RUNUP";
      AN    "HOLDSPD";
      A     "TEMP5";
      A     "VBALM";
      =     "RUNTHRU";
NETWORK
TITLE = RUNTHRUT=(TEMP5)(VBALM)
      A     "TEMP5";
      A     "VBALM";
      =     "RUNTHRUT";
NETWORK
TITLE = RBOSCL=PULSE[NOT{(~VRSCNP)(RUNUP+RUNTHRU)}]
      A(;
      O     "RUNUP";
      O     "RUNTHRU";
      );
      AN    "VRSCNP";
      NOT;
      L     "ATCTime_VALs".T8PULSE;
      SP    T 8;
      NOP   0;
      NOP   0;
      NOP   0;
      A     T 8;
      =     "RBOSCL";
NETWORK
TITLE = RBOS=FF[{(VBALM)(RUNBACK)},{(~ATC5)+RBOSCL}]
      A     "VBALM";
      A     "RUNBACK";
      S     "RBOS";
      A(;
      ON    "ATC5";
      O     "RBOSCL";
      );
      R     "RBOS";
      A     "RBOS";
      =     "RBOS";
NETWORK
TITLE = GORUNUP=FF[RUNBACK,(TEMP5+RUNTHRU)]
      A     "RUNBACK";
      S     "GORUNUP";
      A(;
      O     "TEMP5";
      O     "RUNTHRU";
      );
      R     "GORUNUP";
      A     "GORUNUP";
      =     "GORUNUP";
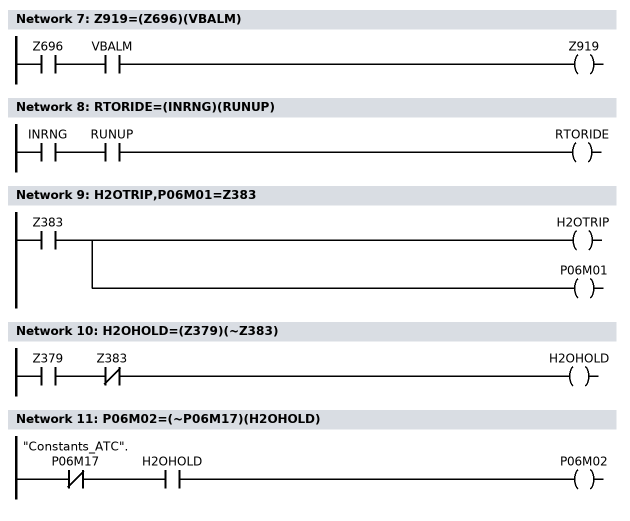
NETWORK
TITLE = Z919=(Z696)(VBALM)
      A     "Z696";
      A     "VBALM";
      =     "Z919";
NETWORK
TITLE = RTORIDE=(INRNG)(RUNUP)
      A     "INRNG";
      A     "RUNUP";
      =     "RTORIDE";
NETWORK
TITLE = H2OTRIP,P06M01=Z383
      A     "Z383";
      =     "H2OTRIP";
      =     "P06M01";
NETWORK
TITLE = H2OHOLD=(Z379)(~Z383)
      A     "Z379";
      AN    "Z383";
      =     "H2OHOLD";
NETWORK
TITLE = P06M02=(~P06M17)(H2OHOLD)
      AN    "Constants_ATC".P06M17;
      A     "H2OHOLD";
      =     "P06M02";
END_FUNCTION

FUNCTION "Sheet 29 (ATC)" : VOID	// FC 110
TITLE = Sheet 29 (ATC)
//VIBRATION RUN THRU REF (Analog)
AUTHOR : RJ
FAMILY : ATC
VERSION : 0.1
BEGIN
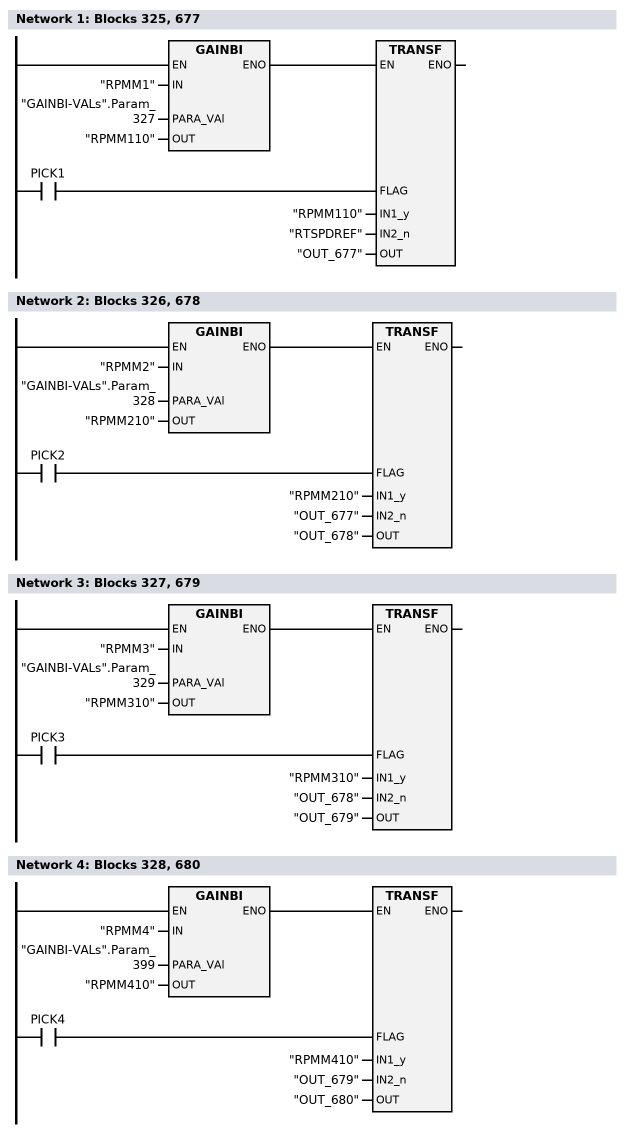
NETWORK
TITLE = Blocks 325, 677
      A     "PICK1";
      =     L 0.0;
      BLD   103;
      A(;
      CALL  "GAINBI" (
           IN                       := "RPMM1",
           PARA_VAl                 := "GAINBI-VALs".Param_327,
           OUT                      := "RPMM110");
      A     BR;
      );
      JNB   _001;
      CALL  "TRANSF" (
           FLAG                     := L 0.0,
           IN1_y                    := "RPMM110",
           IN2_n                    := "RTSPDREF",
           OUT                      := "OUT_677");
_001: NOP   0;
NETWORK
TITLE = Blocks 326, 678
      A     "PICK2";
      =     L 0.0;
      BLD   103;
      A(;
      CALL  "GAINBI" (
           IN                       := "RPMM2",
           PARA_VAl                 := "GAINBI-VALs".Param_328,
           OUT                      := "RPMM210");
      A     BR;
      );
      JNB   _002;
      CALL  "TRANSF" (
           FLAG                     := L 0.0,
           IN1_y                    := "RPMM210",
           IN2_n                    := "OUT_677",
           OUT                      := "OUT_678");
_002: NOP   0;
NETWORK
TITLE = Blocks 327, 679
      A     "PICK3";
      =     L 0.0;
      BLD   103;
      A(;
      CALL  "GAINBI" (
           IN                       := "RPMM3",
           PARA_VAl                 := "GAINBI-VALs".Param_329,
           OUT                      := "RPMM310");
      A     BR;
      );
      JNB   _003;
      CALL  "TRANSF" (
           FLAG                     := L 0.0,
           IN1_y                    := "RPMM310",
           IN2_n                    := "OUT_678",
           OUT                      := "OUT_679");
_003: NOP   0;
NETWORK
TITLE = Blocks 328, 680
      A     "PICK4";
      =     L 0.0;
      BLD   103;
      A(;
      CALL  "GAINBI" (
           IN                       := "RPMM4",
           PARA_VAl                 := "GAINBI-VALs".Param_399,
           OUT                      := "RPMM410");
      A     BR;
      );
      JNB   _004;
      CALL  "TRANSF" (
           FLAG                     := L 0.0,
           IN1_y                    := "RPMM410",
           IN2_n                    := "OUT_679",
           OUT                      := "OUT_680");
_004: NOP   0;
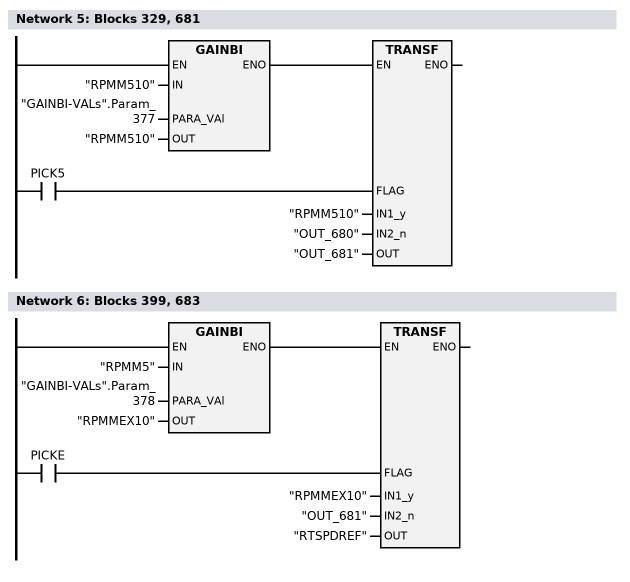
NETWORK
TITLE = Blocks 329, 681
      A     "PICK5";
      =     L 0.0;
      BLD   103;
      A(;
      CALL  "GAINBI" (
           IN                       := "RPMM510",
           PARA_VAl                 := "GAINBI-VALs".Param_377,
           OUT                      := "RPMM510");
      A     BR;
      );
      JNB   _005;
      CALL  "TRANSF" (
           FLAG                     := L 0.0,
           IN1_y                    := "RPMM510",
           IN2_n                    := "OUT_680",
           OUT                      := "OUT_681");
_005: NOP   0;
NETWORK
TITLE = Blocks 399, 683
      A     "PICKE";
      =     L 0.0;
      BLD   103;
      A(;
      CALL  "GAINBI" (
           IN                       := "RPMM5",
           PARA_VAl                 := "GAINBI-VALs".Param_378,
           OUT                      := "RPMMEX10");
      A     BR;
      );
      JNB   _006;
      CALL  "TRANSF" (
           FLAG                     := L 0.0,
           IN1_y                    := "RPMMEX10",
           IN2_n                    := "OUT_681",
           OUT                      := "RTSPDREF");
_006: NOP   0;
END_FUNCTION

FUNCTION "Sheet 30 (ATC)" : VOID	// FC 111
TITLE = Sheet 30 (ATC)
//VIBRATION SPEED REF (Analog)
AUTHOR : RJ
FAMILY : ATC
VERSION : 0.1
BEGIN
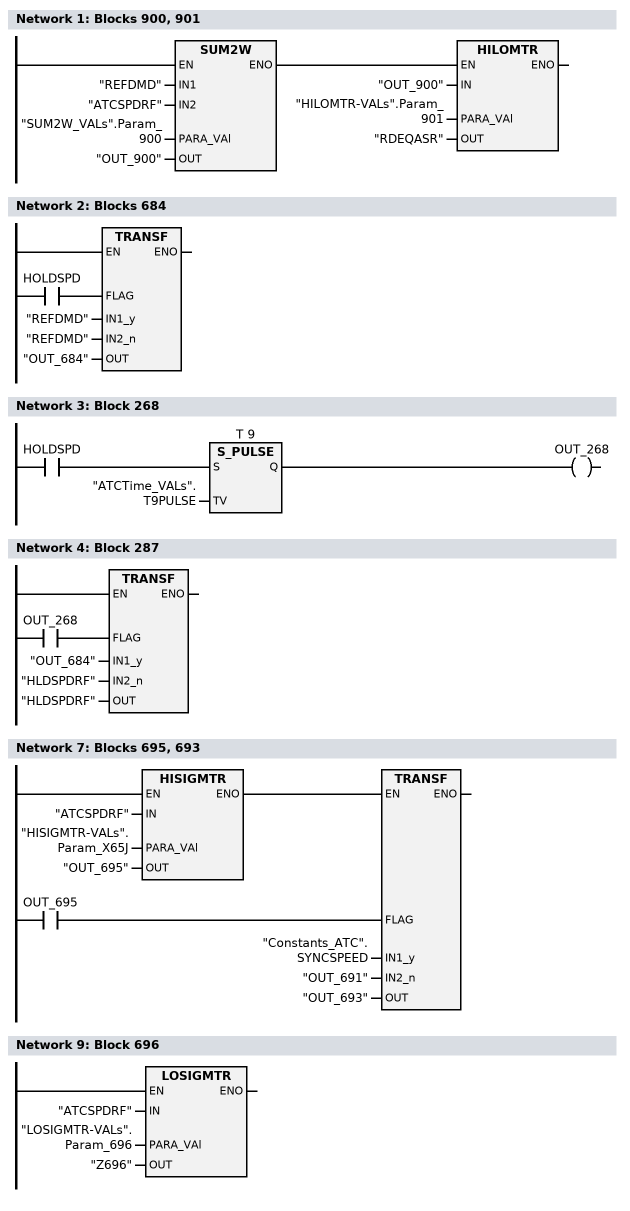
NETWORK
TITLE = Blocks 900, 901 
      A(;
      CALL  "SUM2W" (
           IN1                      := "REFDMD",
           IN2                      := "ATCSPDRF",
           PARA_VAl                 := "SUM2W_VALs".Param_900,
           OUT                      := "OUT_900");
      A     BR;
      );
      JNB   _001;
      CALL  "HILOMTR" (
           IN                       := "OUT_900",
           PARA_VAl                 := "HILOMTR-VALs".Param_901,
           OUT                      := "RDEQASR");
_001: NOP   0;
NETWORK
TITLE = Blocks 684
      A     "HOLDSPD";
      =     L 0.0;
      BLD   103;
      CALL  "TRANSF" (
           FLAG                     := L 0.0,
           IN1_y                    := "REFDMD",
           IN2_n                    := "REFDMD",
           OUT                      := "OUT_684");
      NOP   0;
NETWORK
TITLE = Block 268
      A     "HOLDSPD";
      L     "ATCTime_VALs".T9PULSE;
      SP    T 9;
      NOP   0;
      NOP   0;
      NOP   0;
      A     T 9;
      =     "OUT_268";
NETWORK
TITLE = Block 287
      A     "OUT_268";
      =     L 0.0;
      BLD   103;
      CALL  "TRANSF" (
           FLAG                     := L 0.0,
           IN1_y                    := "OUT_684",
           IN2_n                    := "HLDSPDRF",
           OUT                      := "HLDSPDRF");
      NOP   0;
NETWORK
TITLE = Blocks 687, 688, 689
      A     "RUNTHRU";
      =     L 0.0;
      BLD   103;
      A(;
      A     "RUNDOWN";
      =     L 0.1;
      BLD   103;
      A(;
      A     "RUNUP";
      =     L 0.2;
      BLD   103;
      CALL  "TRANSF" (
           FLAG                     := L 0.2,
           IN1_y                    := "RUSPDREF",
           IN2_n                    := "ATCSPDRF",
           OUT                      := "OUT_687");
      A     BR;
      );
      JNB   _002;
      CALL  "TRANSF" (
           FLAG                     := L 0.1,
           IN1_y                    := "RDSPDREF",
           IN2_n                    := "OUT_687",
           OUT                      := "OUT_688");
_002: A     BR;
      );
      JNB   _003;
      CALL  "TRANSF" (
           FLAG                     := L 0.0,
           IN1_y                    := "RTSPDREF",
           IN2_n                    := "OUT_688",
           OUT                      := "OUT_689");
_003: NOP   0;
NETWORK
TITLE = Blocks 690, 691
      A     "HOLDSPD";
      =     L 0.0;
      BLD   103;
      A(;
      A     "RUNBACK";
      =     L 0.1;
      BLD   103;
      CALL  "TRANSF" (
           FLAG                     := L 0.1,
           IN1_y                    := "RBSPDREF",
           IN2_n                    := "OUT_689",
           OUT                      := "OUT_690");
      A     BR;
      );
      JNB   _004;
      CALL  "TRANSF" (
           FLAG                     := L 0.0,
           IN1_y                    := "HLDSPDRF",
           IN2_n                    := "OUT_690",
           OUT                      := "OUT_691");
_004: NOP   0;
NETWORK
TITLE = Blocks 695, 693
      A     "OUT_695";
      =     L 0.0;
      BLD   103;
      A(;
      CALL  "HISIGMTR" (
           IN                       := "ATCSPDRF",
           PARA_VAl                 := "HISIGMTR-VALs".Param_X65J,
           OUT                      := "OUT_695");
      A     BR;
      );
      JNB   _005;
      CALL  "TRANSF" (
           FLAG                     := L 0.0,
           IN1_y                    := "Constants_ATC".SYNCSPEED,
           IN2_n                    := "OUT_691",
           OUT                      := "OUT_693");
_005: NOP   0;
NETWORK
TITLE = Blocks 694, 994
      A(;
      A(;
      A(;
      A     "Z919";
      =     L 0.0;
      BLD   103;
      CALL  "TRANSF" (
           FLAG                     := L 0.0,
           IN1_y                    := "Z995",
           IN2_n                    := "OUT_693",
           OUT                      := "OUT_694");
      A     BR;
      );
      JNB   _006;
      L     "Constants_ATC".SYNCSPEED;
      T     "HILOLMTV-VALs".Param_994.HILM;
      SET;
      SAVE;
      CLR;
_006: A     BR;
      );
      JNB   _007;
      L     "ATCREFLO";
      T     "HILOLMTV-VALs".Param_994.LOLM;
      SET;
      SAVE;
      CLR;
_007: A     BR;
      );
      JNB   _008;
      CALL  "HILOLMTV" (
           IN                       := "OUT_694",
           PARA_VAl                 := "HILOLMTV-VALs".Param_994,
           OUT                      := "ATCSPDRF");
_008: NOP   0;
NETWORK
TITLE = Block 696
      CALL  "LOSIGMTR" (
           IN                       := "ATCSPDRF",
           PARA_VAl                 := "LOSIGMTR-VALs".Param_696,
           OUT                      := "Z696");
      NOP   0;
END_FUNCTION

FUNCTION "Sheet 31 (ATC)" : VOID	// FC 112
TITLE = Sheet 31 (ATC)
//LOOPS 18, 19. WATER DETECTION (Analog)
AUTHOR : RJ
FAMILY : ATC
VERSION : 0.1
BEGIN
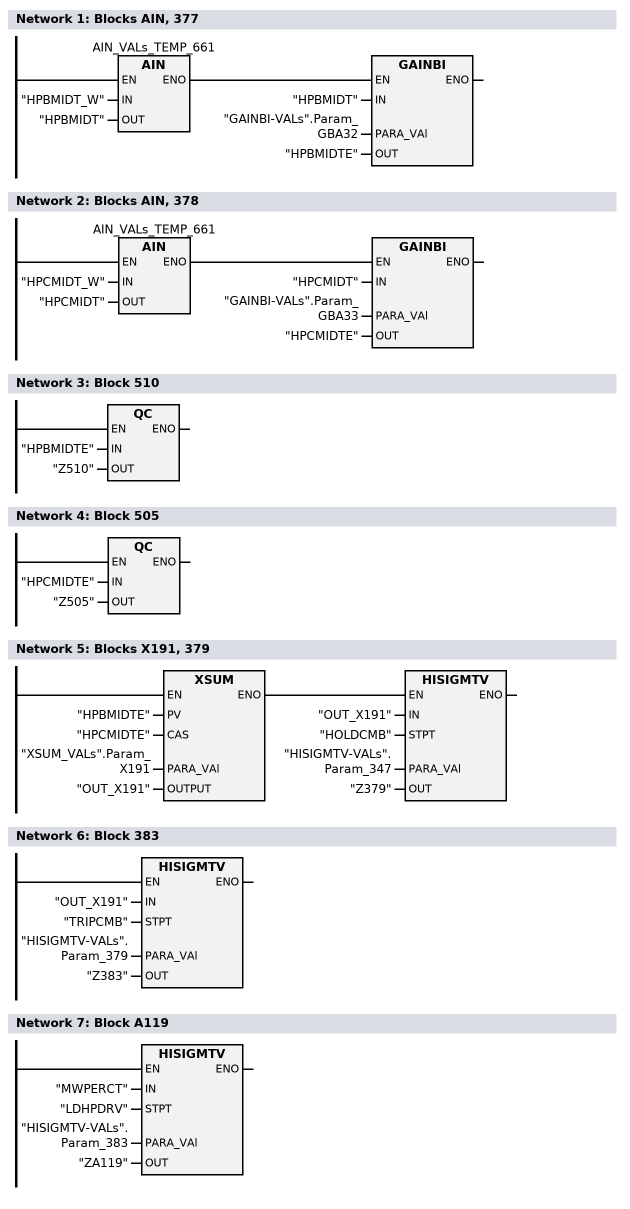
NETWORK
TITLE = Blocks AIN, 377
      A(;
      CALL  "AIN" , "AIN_VALs_TEMP_661" (
           IN                       := "HPBMIDT_W",
           OUT                      := "HPBMIDT");
      A     BR;
      );
      JNB   _001;
      CALL  "GAINBI" (
           IN                       := "HPBMIDT",
           PARA_VAl                 := "GAINBI-VALs".Param_GBA32,
           OUT                      := "HPBMIDTE");
_001: NOP   0;
NETWORK
TITLE = Blocks AIN, 378
      A(;
      CALL  "AIN" , "AIN_VALs_TEMP_661" (
           IN                       := "HPCMIDT_W",
           OUT                      := "HPCMIDT");
      A     BR;
      );
      JNB   _002;
      CALL  "GAINBI" (
           IN                       := "HPCMIDT",
           PARA_VAl                 := "GAINBI-VALs".Param_GBA33,
           OUT                      := "HPCMIDTE");
_002: NOP   0;
NETWORK
TITLE = Block 510
      CALL  "QC" (
           IN                       := "HPBMIDTE",
           OUT                      := "Z510");
      NOP   0;
NETWORK
TITLE = Block 505
      CALL  "QC" (
           IN                       := "HPCMIDTE",
           OUT                      := "Z505");
      NOP   0;
NETWORK
TITLE = Blocks X191, 379
      A(;
      CALL  "XSUM" (
           PV                       := "HPBMIDTE",
           CAS                      := "HPCMIDTE",
           PARA_VAl                 := "XSUM_VALs".Param_X191,
           OUTPUT                   := "OUT_X191");
      A     BR;
      );
      JNB   _003;
      CALL  "HISIGMTV" (
           IN                       := "OUT_X191",
           STPT                     := "HOLDCMB",
           PARA_VAl                 := "HISIGMTV-VALs".Param_347,
           OUT                      := "Z379");
_003: NOP   0;
NETWORK
TITLE = Block 383
      CALL  "HISIGMTV" (
           IN                       := "OUT_X191",
           STPT                     := "TRIPCMB",
           PARA_VAl                 := "HISIGMTV-VALs".Param_379,
           OUT                      := "Z383");
      NOP   0;
NETWORK
TITLE = Block A119
      CALL  "HISIGMTV" (
           IN                       := "MWPERCT",
           STPT                     := "LDHPDRV",
           PARA_VAl                 := "HISIGMTV-VALs".Param_383,
           OUT                      := "ZA119");
      NOP   0;
END_FUNCTION

FUNCTION "Sheet 32 (ATC)" : VOID	// FC 113
TITLE = Sheet 32 (ATC)
//LADDERS 49, 51, 53. DRAIN VALVE LOGIC (Digital)
AUTHOR : RJ
FAMILY : ATC
VERSION : 0.1
BEGIN
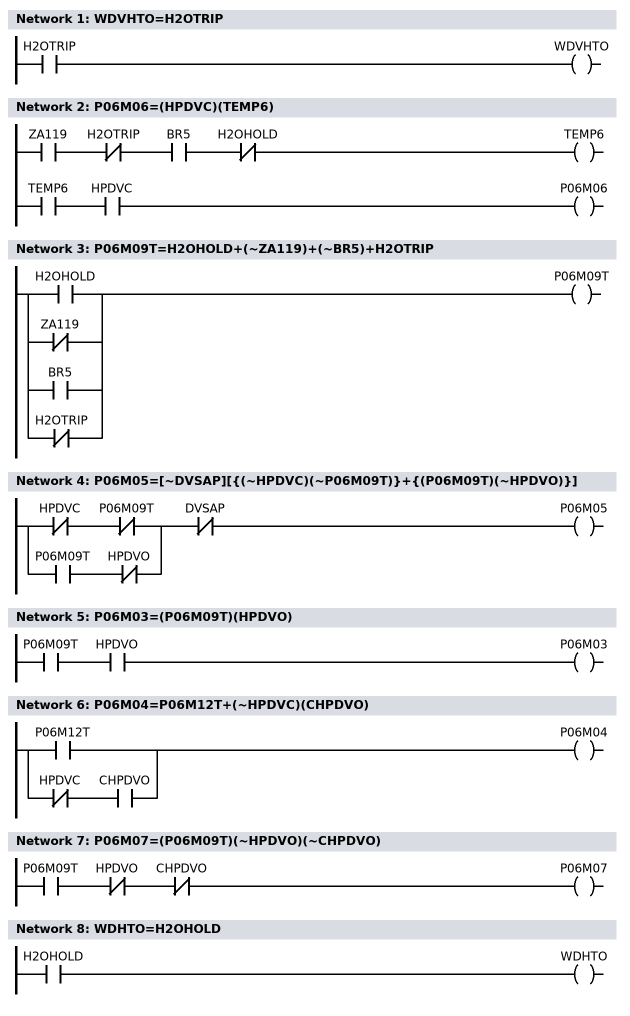
NETWORK
TITLE = WDVHTO=H2OTRIP
      A     "H2OTRIP";
      =     "WDVHTO";
NETWORK
TITLE = P06M06=(HPDVC)(TEMP6)
//TEMP6=(Z119)(~H2OTRIP)(BR5)(~H2OHOLD)
      A     "ZA119";
      AN    "H2OTRIP";
      A     "BR5";
      AN    "H2OHOLD";
      =     "TEMP6";
      A     "TEMP6";
      A     "HPDVC";
      =     "P06M06";
NETWORK
TITLE = P06M09T=H2OHOLD+(~ZA119)+(~BR5)+H2OTRIP
      O     "H2OHOLD";
      ON    "ZA119";
      O     "BR5";
      ON    "H2OTRIP";
      =     "P06M09T";
NETWORK
TITLE = P06M05=[~DVSAP][{(~HPDVC)(~P06M09T)}+{(P06M09T)(~HPDVO)}]
      A(;
      AN    "HPDVC";
      AN    "P06M09T";
      O;
      A     "P06M09T";
      AN    "HPDVO";
      );
      AN    "DVSAP";
      =     "P06M05";
NETWORK
TITLE = P06M03=(P06M09T)(HPDVO)
      A     "P06M09T";
      A     "HPDVO";
      =     "P06M03";
NETWORK
TITLE = P06M04=P06M12T+(~HPDVC)(CHPDVO)
      O     "P06M12T";
      O;
      AN    "HPDVC";
      A     "CHPDVO";
      =     "P06M04";
NETWORK
TITLE = P06M07=(P06M09T)(~HPDVO)(~CHPDVO)
      A     "P06M09T";
      AN    "HPDVO";
      AN    "CHPDVO";
      =     "P06M07";
NETWORK
TITLE = WDHTO=H2OHOLD
      A     "H2OHOLD";
      =     "WDHTO";
END_FUNCTION

// FC 115: know-how protected block, not included

FUNCTION "SUBB24" : VOID	// FC 116
TITLE = SUBB24
//Supporting block for sheet 24 (ATC)
AUTHOR : RJ
FAMILY : ATC
VERSION : 0.1
VAR_INPUT
  VBABS : REAL ;
  VBTRIP : REAL ;
  IN_SUM2W1 : UDT 12;
  IN_GAINBI : UDT 4;
  IN_SUM2W2 : UDT 12;
  IN_HISIGMTV : UDT 8;
  IN_HISIGMTR : UDT 1;
END_VAR
VAR_OUTPUT
  APVBTP : BOOL ;
  VBINC : BOOL ;
END_VAR
VAR_TEMP
  VBDIFF : REAL ;
  VBTMP : REAL ;
  VBANT : REAL ;
  VBP : REAL ;
  Param_SUM2W2 : UDT 12;
  Param_SUM2W1 : UDT 12;
  Param_GAINBI : UDT 4;
  Param_HISIGMTR : UDT 1;
  Param_HISIGMTV : UDT 8;
END_VAR
BEGIN
NETWORK
TITLE = SUM2W1
      A(;
      BLD   5;
      T     LD 54;
      TAK;
      T     LD 58;
      L     P##IN_SUM2W1;
      LAR1;
      L     W [AR1,P#0.0];
      T     LW 52;
      OPN   DB [LW 52];
      L     D [AR1,P#2.0];
      LAR1;
      L     LD 58;
      L     LD 54;
      L     D [AR1,P#0.0];
      T     #Param_SUM2W1.WT1;
      SET;
      SAVE;
      CLR;
      A     BR;
      );
      JNB   _001;
      BLD   5;
      T     LD 54;
      TAK;
      T     LD 58;
      L     P##IN_SUM2W1;
      LAR1;
      L     W [AR1,P#0.0];
      T     LW 52;
      OPN   DB [LW 52];
      L     D [AR1,P#2.0];
      LAR1;
      L     LD 58;
      L     LD 54;
      L     D [AR1,P#4.0];
      T     #Param_SUM2W1.WT2;
_001: NOP   0;
NETWORK
TITLE = SUM2W2
      A(;
      BLD   5;
      T     LD 54;
      TAK;
      T     LD 58;
      L     P##IN_SUM2W2;
      LAR1;
      L     W [AR1,P#0.0];
      T     LW 52;
      OPN   DB [LW 52];
      L     D [AR1,P#2.0];
      LAR1;
      L     LD 58;
      L     LD 54;
      L     D [AR1,P#0.0];
      T     #Param_SUM2W2.WT1;
      SET;
      SAVE;
      CLR;
      A     BR;
      );
      JNB   _002;
      BLD   5;
      T     LD 54;
      TAK;
      T     LD 58;
      L     P##IN_SUM2W2;
      LAR1;
      L     W [AR1,P#0.0];
      T     LW 52;
      OPN   DB [LW 52];
      L     D [AR1,P#2.0];
      LAR1;
      L     LD 58;
      L     LD 54;
      L     D [AR1,P#4.0];
      T     #Param_SUM2W2.WT2;
_002: NOP   0;
NETWORK
TITLE = GAINBI
      A(;
      BLD   5;
      T     LD 54;
      TAK;
      T     LD 58;
      L     P##IN_GAINBI;
      LAR1;
      L     W [AR1,P#0.0];
      T     LW 52;
      OPN   DB [LW 52];
      L     D [AR1,P#2.0];
      LAR1;
      L     LD 58;
      L     LD 54;
      L     D [AR1,P#4.0];
      T     #Param_GAINBI.BIAS;
      SET;
      SAVE;
      CLR;
      A     BR;
      );
      JNB   _003;
      BLD   5;
      T     LD 54;
      TAK;
      T     LD 58;
      L     P##IN_GAINBI;
      LAR1;
      L     W [AR1,P#0.0];
      T     LW 52;
      OPN   DB [LW 52];
      L     D [AR1,P#2.0];
      LAR1;
      L     LD 58;
      L     LD 54;
      L     D [AR1,P#0.0];
      T     #Param_GAINBI.GAIN;
_003: NOP   0;
NETWORK
TITLE = HISIGMTR
      A(;
      BLD   5;
      T     LD 54;
      TAK;
      T     LD 58;
      L     P##IN_HISIGMTR;
      LAR1;
      L     W [AR1,P#0.0];
      T     LW 52;
      OPN   DB [LW 52];
      L     D [AR1,P#2.0];
      LAR1;
      L     LD 58;
      L     LD 54;
      L     D [AR1,P#4.0];
      T     #Param_HISIGMTR.DBAN;
      SET;
      SAVE;
      CLR;
      A     BR;
      );
      JNB   _004;
      BLD   5;
      T     LD 54;
      TAK;
      T     LD 58;
      L     P##IN_HISIGMTR;
      LAR1;
      L     W [AR1,P#0.0];
      T     LW 52;
      OPN   DB [LW 52];
      L     D [AR1,P#2.0];
      LAR1;
      L     LD 58;
      L     LD 54;
      L     D [AR1,P#0.0];
      T     #Param_HISIGMTR.STPT;
_004: NOP   0;
NETWORK
TITLE = HISIGMTV
      BLD   5;
      T     LD 54;
      TAK;
      T     LD 58;
      L     P##IN_HISIGMTV;
      LAR1;
      L     W [AR1,P#0.0];
      T     LW 52;
      OPN   DB [LW 52];
      L     D [AR1,P#2.0];
      LAR1;
      L     LD 58;
      L     LD 54;
      L     D [AR1,P#0.0];
      T     #Param_HISIGMTV;
      NOP   0;
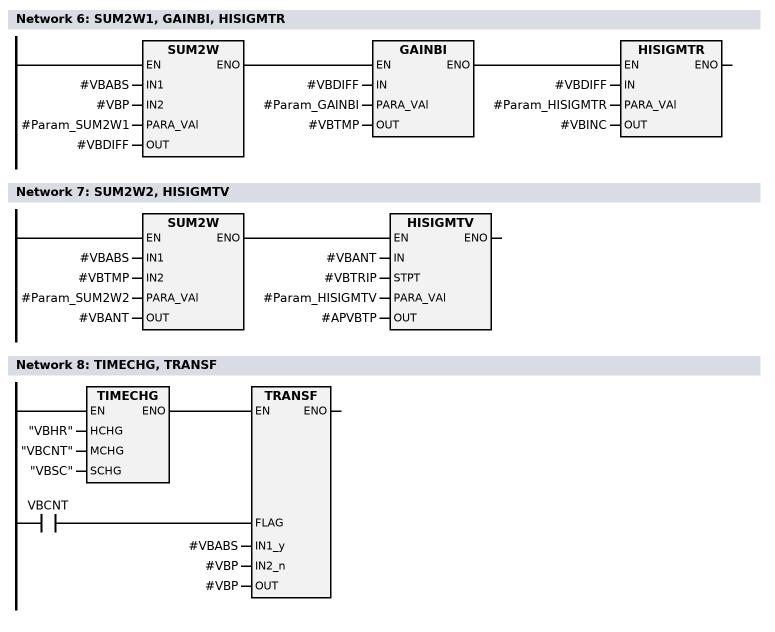
NETWORK
TITLE = SUM2W1, GAINBI, HISIGMTR
      A(;
      A(;
      CALL  "SUM2W" (
           IN1                      := #VBABS,
           IN2                      := #VBP,
           PARA_VAl                 := #Param_SUM2W1,
           OUT                      := #VBDIFF);
      A     BR;
      );
      JNB   _005;
      CALL  "GAINBI" (
           IN                       := #VBDIFF,
           PARA_VAl                 := #Param_GAINBI,
           OUT                      := #VBTMP);
_005: A     BR;
      );
      JNB   _006;
      CALL  "HISIGMTR" (
           IN                       := #VBDIFF,
           PARA_VAl                 := #Param_HISIGMTR,
           OUT                      := #VBINC);
_006: NOP   0;
NETWORK
TITLE = SUM2W2, HISIGMTV
      A(;
      CALL  "SUM2W" (
           IN1                      := #VBABS,
           IN2                      := #VBTMP,
           PARA_VAl                 := #Param_SUM2W2,
           OUT                      := #VBANT);
      A     BR;
      );
      JNB   _007;
      CALL  "HISIGMTV" (
           IN                       := #VBANT,
           STPT                     := #VBTRIP,
           PARA_VAl                 := #Param_HISIGMTV,
           OUT                      := #APVBTP);
_007: NOP   0;
NETWORK
TITLE = TIMECHG, TRANSF
      A     "VBCNT";
      =     L 52.0;
      BLD   103;
      A(;
      CALL  "TIMECHG" (
           HCHG                     := "VBHR",
           MCHG                     := "VBCNT",
           SCHG                     := "VBSC");
      A     BR;
      );
      JNB   _008;
      CALL  "TRANSF" (
           FLAG                     := L 52.0,
           IN1_y                    := #VBABS,
           IN2_n                    := #VBP,
           OUT                      := #VBP);
_008: NOP   0;
END_FUNCTION

FUNCTION "TIMECHG" : VOID	// FC 117
TITLE = TIMECHG
//Check Real-Time Clock, Set Flags
AUTHOR : RJ
VERSION : 0.1
VAR_OUTPUT
  HCHG : BOOL ;
  MCHG : BOOL ;
  SCHG : BOOL ;
END_VAR
VAR_TEMP
  CDT : DATE_AND_TIME ;
  RET : INT ;
  CTIME : TIME_OF_DAY ;
  H : INT ;
  M : INT ;
  S : INT ;
END_VAR
BEGIN
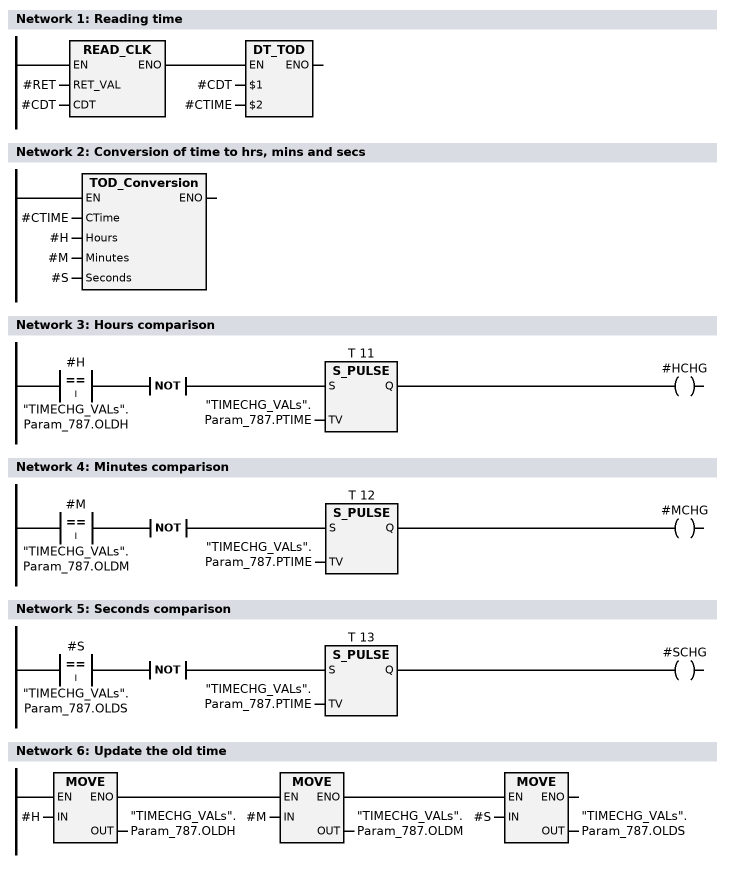
NETWORK
TITLE = Reading time
      A(;
      CALL  "READ_CLK" (
           RET_VAL                  := #RET,
           CDT                      := #CDT);
      A     BR;
      );
      JNB   _001;
      CALL  "DT_TOD" (
           $1                       := #CDT,
           $2                       := #CTIME);
_001: NOP   0;
NETWORK
TITLE = Conversion of time to hrs, mins and secs
      CALL  "TOD_Conversion" (
           CTime                    := #CTIME,
           Hours                    := #H,
           Minutes                  := #M,
           Seconds                  := #S);
      NOP   0;
NETWORK
TITLE = Hours comparison
      A(;
      L     #H;
      L     "TIMECHG_VALs".Param_787.OLDH;
      ==I;
      );
      NOT;
      L     "TIMECHG_VALs".Param_787.PTIME;
      SP    T 11;
      NOP   0;
      NOP   0;
      NOP   0;
      A     T 11;
      =     #HCHG;
NETWORK
TITLE = Minutes comparison
      A(;
      L     #M;
      L     "TIMECHG_VALs".Param_787.OLDM;
      ==I;
      );
      NOT;
      L     "TIMECHG_VALs".Param_787.PTIME;
      SP    T 12;
      NOP   0;
      NOP   0;
      NOP   0;
      A     T 12;
      =     #MCHG;
NETWORK
TITLE = Seconds comparison
      A(;
      L     #S;
      L     "TIMECHG_VALs".Param_787.OLDS;
      ==I;
      );
      NOT;
      L     "TIMECHG_VALs".Param_787.PTIME;
      SP    T 13;
      NOP   0;
      NOP   0;
      NOP   0;
      A     T 13;
      =     #SCHG;
NETWORK
TITLE = Update the old time
      A(;
      A(;
      L     #H;
      T     "TIMECHG_VALs".Param_787.OLDH;
      SET;
      SAVE;
      CLR;
      A     BR;
      );
      JNB   _002;
      L     #M;
      T     "TIMECHG_VALs".Param_787.OLDM;
      SET;
      SAVE;
      CLR;
_002: A     BR;
      );
      JNB   _003;
      L     #S;
      T     "TIMECHG_VALs".Param_787.OLDS;
_003: NOP   0;
END_FUNCTION

FUNCTION "Sheet 33 (ATC)" : VOID	// FC 118
TITLE = Sheet 33 (ATC)
//LOOPS 4, 5 (Analog)
AUTHOR : RJ
FAMILY : ATC
VERSION : 0.1
BEGIN
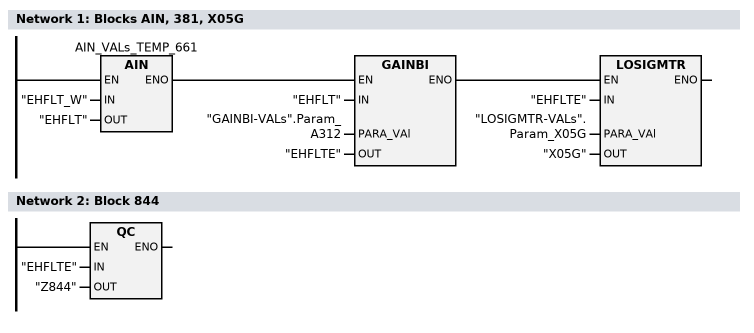
NETWORK
TITLE = Blocks AIN, 381, X05G
      A(;
      A(;
      CALL  "AIN" , "AIN_VALs_TEMP_661" (
           IN                       := "EHFLT_W",
           OUT                      := "EHFLT");
      A     BR;
      );
      JNB   _001;
      CALL  "GAINBI" (
           IN                       := "EHFLT",
           PARA_VAl                 := "GAINBI-VALs".Param_A312,
           OUT                      := "EHFLTE");
_001: A     BR;
      );
      JNB   _002;
      CALL  "LOSIGMTR" (
           IN                       := "EHFLTE",
           PARA_VAl                 := "LOSIGMTR-VALs".Param_X05G,
           OUT                      := "X05G");
_002: NOP   0;
NETWORK
TITLE = Block 844
      CALL  "QC" (
           IN                       := "EHFLTE",
           OUT                      := "Z844");
      NOP   0;
END_FUNCTION

FUNCTION "Sheet 34 (ATC)" : VOID	// FC 119
TITLE = Sheet 34 (ATC)
//LADDERS 19, 21, 23, 25, 27. TURNING GEAR - P03MXX (Digital)
AUTHOR : RJ
FAMILY : ATC
VERSION : 0.1
BEGIN
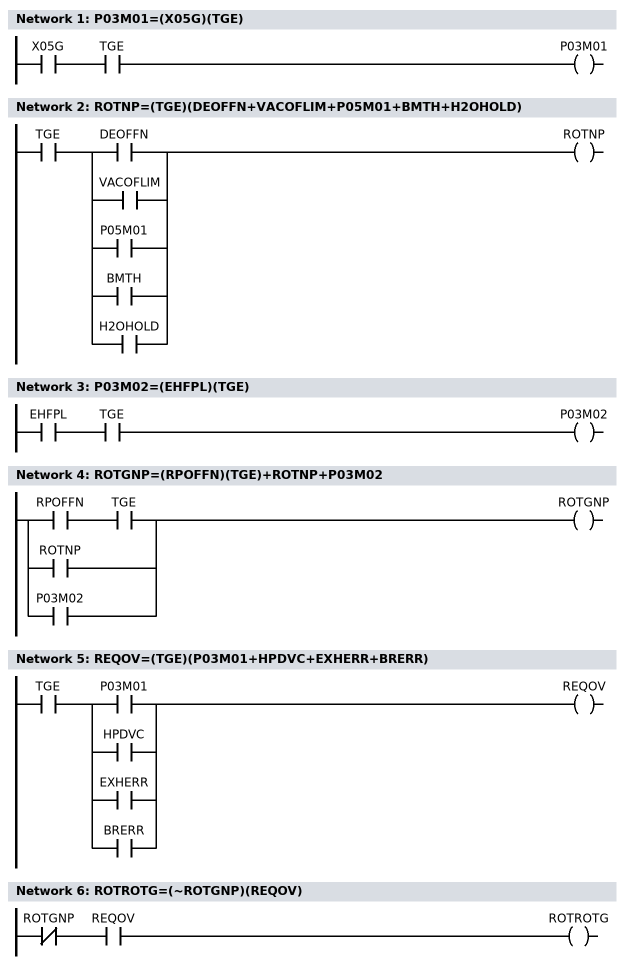
NETWORK
TITLE = P03M01=(X05G)(TGE)
      A     "X05G";
      A     "TGE";
      =     "P03M01";
NETWORK
TITLE = ROTNP=(TGE)(DEOFFN+VACOFLIM+P05M01+BMTH+H2OHOLD)
      A     "TGE";
      A(;
      O     "DEOFFN";
      O     "VACOFLIM";
      O     "P05M01";
      O     "BMTH";
      O     "H2OHOLD";
      );
      =     "ROTNP";
NETWORK
TITLE = P03M02=(EHFPL)(TGE)
      A     "EHFPL";
      A     "TGE";
      =     "P03M02";
NETWORK
TITLE = ROTGNP=(RPOFFN)(TGE)+ROTNP+P03M02
      A     "RPOFFN";
      A     "TGE";
      O     "ROTNP";
      O     "P03M02";
      =     "ROTGNP";
NETWORK
TITLE = REQOV=(TGE)(P03M01+HPDVC+EXHERR+BRERR)
      A     "TGE";
      A(;
      O     "P03M01";
      O     "HPDVC";
      O     "EXHERR";
      O     "BRERR";
      );
      =     "REQOV";
NETWORK
TITLE = ROTROTG=(~ROTGNP)(REQOV)
      AN    "ROTGNP";
      A     "REQOV";
      =     "ROTROTG";
END_FUNCTION

FUNCTION "Sheet 35 (ATC)" : VOID	// FC 120
TITLE = Sheet 35 (ATC)
//LOOPS 6, 60. THRUST BEARING, ROTOR ECCEN. (Analog)
AUTHOR : RJ
FAMILY : ATC
VERSION : 0.1
BEGIN
